LIN {X 0,Y 279.122,Z 639.162,A -85,B 0,C 180,E1 -18844.948,E2 -18844.948} C_VEL
LIN {X 0,Y 285.819,Z 626.252,A -85,B 0,C 180,E1 -18847.044,E2 -18847.044} C_VEL
LIN {X 0,Y 292.614,Z 612.071,A -85,B 0,C 180,E1 -18848.864,E2 -18848.864} C_VEL
LIN {X 0,Y 299.456,Z 596.451,A -85,B 0,C 180,E1 -18850.417,E2 -18850.417} C_VEL
LIN {X 0,Y 305.025,Z 582.195,A -85,B 0,C 180,E1 -18851.485,E2 -18851.485} C_VEL
LIN {X 0,Y 310.133,Z 566.91,A -85,B 0,C 180,E1 -18852.39,E2 -18852.39} C_VEL
LIN {X 0,Y 315.424,Z 547.486,A -85,B 0,C 180,E1 -18853.247,E2 -18853.247} C_VEL
LIN {X 0,Y 330.429,Z 486.43,A -85,B 0,C 180,E1 -18855.632,E2 -18855.632} C_VEL
LIN {X 0,Y 330.312,Z 486.665,A -85,B 0,C 180,E1 -18857.244,E2 -18857.244} C_VEL
LIN {X 0,Y 313.368,Z 553.571,A -85,B 0,C 180,E1 -18860.061,E2 -18860.061} C_VEL
LIN {X 0,Y 309.554,Z 566.236,A -85,B 0,C 180,E1 -18860.738,E2 -18860.738} C_VEL
LIN {X 0,Y 304.046,Z 581.734,A -85,B 0,C 180,E1 -18861.849,E2 -18861.849} C_VEL
LIN {X 0,Y 298.06,Z 596.489,A -85,B 0,C 180,E1 -18863.25,E2 -18863.25} C_VEL
LIN {X 0,Y 292.263,Z 609.131,A -85,B 0,C 180,E1 -18864.752,E2 -18864.752} C_VEL
LIN {X 0,Y 286.298,Z 620.873,A -85,B 0,C 180,E1 -18866.473,E2 -18866.473} C_VEL
LIN {X 0,Y 279.847,Z 632.628,A -85,B 0,C 180,E1 -18868.635,E2 -18868.635} C_VEL
LIN {X 0,Y 273.436,Z 643.529,A -85,B 0,C 180,E1 -18871.189,E2 -18871.189} C_VEL
LIN {X 0,Y 267.673,Z 652.584,A -85,B 0,C 180,E1 -18873.91,E2 -18873.91} C_VEL
LIN {X 0,Y 263.097,Z 659.179,A -85,B 0,C 180,E1 -18876.379,E2 -18876.379} C_VEL
LIN {X 0,Y 258.649,Z 665.21,A -85,B 0,C 180,E1 -18879.315,E2 -18879.315} C_VEL
LIN {X 0,Y 255.015,Z 669.8,A -85,B 0,C 180,E1 -18882.353,E2 -18882.353} C_VEL
LIN {X 0,Y 252.199,Z 673.017,A -85,B 0,C 180,E1 -18885.475,E2 -18885.475} C_VEL
LIN {X 0,Y 250.06,Z 674.932,A -85,B 0,C 180,E1 -18888.654,E2 -18888.654} C_VEL
LIN {X 0,Y 248.52,Z 675.55,A -85,B 0,C 180,E1 -18891.871,E2 -18891.871} C_VEL
LIN {X 0,Y 247.631,Z 674.837,A -85,B 0,C 180,E1 -18895.116,E2 -18895.116} C_VEL
LIN {X 0,Y 247.2,Z 672.768,A -85,B 0,C 180,E1 -18898.371,E2 -18898.371} C_VEL
LIN {X 0,Y 247.103,Z 669.276,A -85,B 0,C 180,E1 -18901.63,E2 -18901.63} C_VEL
LIN {X 0,Y 247.107,Z 665.658,A -85,B 0,C 180,E1 -18904.078,E2 -18904.078} C_VEL
LIN {X 0,Y 247.454,Z 659.333,A -85,B 0,C 180,E1 -18907.343,E2 -18907.343} C_VEL
LIN {X 0,Y 247.942,Z 652.241,A -85,B 0,C 180,E1 -18910.204,E2 -18910.204} C_VEL
LIN {X 0,Y 248.776,Z 643.485,A -85,B 0,C 180,E1 -18913.062,E2 -18913.062} C_VEL
LIN {X 0,Y 249.849,Z 634.415,A -85,B 0,C 180,E1 -18915.499,E2 -18915.499} C_VEL
LIN {X 0,Y 251.203,Z 623.335,A -85,B 0,C 180,E1 -18917.966,E2 -18917.966} C_VEL
LIN {X 0,Y 252.63,Z 611.516,A -85,B 0,C 180,E1 -18920.137,E2 -18920.137} C_VEL
LIN {X 0,Y 254.248,Z 598.401,A -85,B 0,C 180,E1 -18922.125,E2 -18922.125} C_VEL
LIN {X 0,Y 255.806,Z 585.81,A -85,B 0,C 180,E1 -18923.691,E2 -18923.691} C_VEL
LIN {X 0,Y 257.309,Z 571.28,A -85,B 0,C 180,E1 -18925.155,E2 -18925.155} C_VEL
LIN {X 0,Y 258.67,Z 555.661,A -85,B 0,C 180,E1 -18926.361,E2 -18926.361} C_VEL
LIN {X 0,Y 259.846,Z 539.566,A -85,B 0,C 180,E1 -18927.263,E2 -18927.263} C_VEL
LIN {X 0,Y 265.823,Z 443.881,A -85,B 0,C 180,E1 -18931.363,E2 -18931.363} C_VEL
LIN {X 0,Y 262.638,Z 420.691,A -85,B 0,C 180,E1 -18932.7,E2 -18932.7} C_VEL
LIN {X 0,Y 254.847,Z 398.323,A -85,B 0,C 180,E1 -18934.485,E2 -18934.485} C_VEL
LIN {X 0,Y 252.265,Z 387.318,A -85,B 0,C 180,E1 -18937.963,E2 -18937.963} C_VEL
LIN {X 0,Y 252.455,Z 387.301,A -85,B 0,C 180,E1 -18938.387,E2 -18938.387} C_VEL
LIN {X 0,Y 254.663,Z 388.809,A -85,B 0,C 180,E1 -18939.401,E2 -18939.401} C_VEL
LIN {X 0,Y 256.067,Z 390.357,A -85,B 0,C 180,E1 -18940.164,E2 -18940.164} C_VEL
LIN {X 0,Y 258.345,Z 395.76,A -85,B 0,C 180,E1 -18941.984,E2 -18941.984} C_VEL
LIN {X 0,Y 265.426,Z 407.166,A -85,B 0,C 180,E1 -18944.104,E2 -18944.104} C_VEL
LIN {X 0,Y 272.266,Z 419.25,A -85,B 0,C 180,E1 -18946.001,E2 -18946.001} C_VEL
LIN {X 0,Y 278.453,Z 431.445,A -85,B 0,C 180,E1 -18947.632,E2 -18947.632} C_VEL
LIN {X 0,Y 284.463,Z 445.002,A -85,B 0,C 180,E1 -18949.167,E2 -18949.167} C_VEL
LIN {X 0,Y 285.13,Z 447.431,A -85,B 0,C 180,E1 -18949.361,E2 -18949.361} C_VEL
LIN {X 0,Y 285.914,Z 453.843,A -85,B 0,C 180,E1 -18949.703,E2 -18949.703} C_VEL
LIN {X 0,Y 280.683,Z 561.87,A -85,B 0,C 180,E1 -18952.33,E2 -18952.33} C_VEL
LIN {X 0,Y 279.274,Z 577.479,A -85,B 0,C 180,E1 -18952.902,E2 -18952.902} C_VEL
LIN {X 0,Y 277.366,Z 591.845,A -85,B 0,C 180,E1 -18953.68,E2 -18953.68} C_VEL
LIN {X 0,Y 275.035,Z 605.926,A -85,B 0,C 180,E1 -18954.724,E2 -18954.724} C_VEL
LIN {X 0,Y 272.571,Z 618.27,A -85,B 0,C 180,E1 -18955.888,E2 -18955.888} C_VEL
LIN {X 0,Y 269.432,Z 631.557,A -85,B 0,C 180,E1 -18957.453,E2 -18957.453} C_VEL
LIN {X 0,Y 265.837,Z 644.861,A -85,B 0,C 180,E1 -18959.408,E2 -18959.408} C_VEL
LIN {X 0,Y 262.248,Z 656.841,A -85,B 0,C 180,E1 -18961.596,E2 -18961.596} C_VEL
LIN {X 0,Y 259.213,Z 666.822,A -85,B 0,C 180,E1 -18963.836,E2 -18963.836} C_VEL
LIN {X 0,Y 255.926,Z 676.732,A -85,B 0,C 180,E1 -18966.535,E2 -18966.535} C_VEL
LIN {X 0,Y 253.233,Z 684.89,A -85,B 0,C 180,E1 -18969.277,E2 -18969.277} C_VEL
LIN {X 0,Y 250.896,Z 692.062,A -85,B 0,C 180,E1 -18972.25,E2 -18972.25} C_VEL
LIN {X 0,Y 249.241,Z 697.898,A -85,B 0,C 180,E1 -18975.299,E2 -18975.299} C_VEL
LIN {X 0,Y 247.924,Z 702.738,A -85,B 0,C 180,E1 -18978.554,E2 -18978.554} C_VEL
LIN {X 0,Y 247.181,Z 706.288,A -85,B 0,C 180,E1 -18981.827,E2 -18981.827} C_VEL
LIN {X 0,Y 246.84,Z 708.688,A -85,B 0,C 180,E1 -18985.219,E2 -18985.219} C_VEL
LIN {X 0,Y 246.853,Z 709.819,A -85,B 0,C 180,E1 -18988.368,E2 -18988.368} C_VEL
LIN {X 0,Y 246.854,Z 709.83,A -85,B 0,C 180,E1 -18991.631,E2 -18991.631} C_VEL
LIN {X 0,Y 246.846,Z 708.687,A -85,B 0,C 180,E1 -18994.9,E2 -18994.9} C_VEL
LIN {X 0,Y 247.18,Z 706.393,A -85,B 0,C 180,E1 -18998.173,E2 -18998.173} C_VEL
LIN {X 0,Y 247.908,Z 702.898,A -85,B 0,C 180,E1 -19001.446,E2 -19001.446} C_VEL
LIN {X 0,Y 249.211,Z 698.113,A -85,B 0,C 180,E1 -19004.703,E2 -19004.703} C_VEL
LIN {X 0,Y 250.995,Z 691.907,A -85,B 0,C 180,E1 -19007.939,E2 -19007.939} C_VEL
LIN {X 0,Y 253.499,Z 684.109,A -85,B 0,C 180,E1 -19011.125,E2 -19011.125} C_VEL
LIN {X 0,Y 256.281,Z 675.796,A -85,B 0,C 180,E1 -19013.859,E2 -19013.859} C_VEL
LIN {X 0,Y 259.055,Z 667.491,A -85,B 0,C 180,E1 -19016.118,E2 -19016.118} C_VEL
LIN {X 0,Y 262.148,Z 657.361,A -85,B 0,C 180,E1 -19018.415,E2 -19018.415} C_VEL
LIN {X 0,Y 265.744,Z 645.49,A -85,B 0,C 180,E1 -19020.603,E2 -19020.603} C_VEL
LIN {X 0,Y 268.954,Z 633.613,A -85,B 0,C 180,E1 -19022.39,E2 -19022.39} C_VEL
LIN {X 0,Y 272.096,Z 620.752,A -85,B 0,C 180,E1 -19023.956,E2 -19023.956} C_VEL
LIN {X 0,Y 274.884,Z 607.255,A -85,B 0,C 180,E1 -19025.275,E2 -19025.275} C_VEL
LIN {X 0,Y 277.193,Z 593.324,A -85,B 0,C 180,E1 -19026.345,E2 -19026.345} C_VEL
LIN {X 0,Y 279.272,Z 578.654,A -85,B 0,C 180,E1 -19027.155,E2 -19027.155} C_VEL
LIN {X 0,Y 280.657,Z 563.713,A -85,B 0,C 180,E1 -19027.73,E2 -19027.73} C_VEL
LIN {X 0,Y 284.824,Z 478.026,A -85,B 0,C 180,E1 -19029.833,E2 -19029.833} C_VEL
LIN {X 0,Y 285.995,Z 452.937,A -85,B 0,C 180,E1 -19030.445,E2 -19030.445} C_VEL
LIN {X 0,Y 284.792,Z 445.554,A -85,B 0,C 180,E1 -19030.892,E2 -19030.892} C_VEL
LIN {X 0,Y 277.817,Z 429.915,A -85,B 0,C 180,E1 -19032.679,E2 -19032.679} C_VEL
LIN {X 0,Y 271.176,Z 417.234,A -85,B 0,C 180,E1 -19034.438,E2 -19034.438} C_VEL
LIN {X 0,Y 266.905,Z 409.496,A -85,B 0,C 180,E1 -19035.63,E2 -19035.63} C_VEL
LIN {X 0,Y 262.844,Z 404.965,A -85,B 0,C 180,E1 -19036.739,E2 -19036.739} C_VEL
LIN {X 0,Y 251.385,Z 395.568,A -85,B 0,C 180,E1 -19040.001,E2 -19040.001} C_VEL
LIN {X 0,Y 250.424,Z 394.069,A -85,B 0,C 180,E1 -19040.529,E2 -19040.529} C_VEL
LIN {X 0,Y 246.627,Z 385.224,A -85,B 0,C 180,E1 -19044.026,E2 -19044.026} C_VEL
LIN {X 0,Y 243.811,Z 378.951,A -85,B 0,C 180,E1 -19046.791,E2 -19046.791} C_VEL
LIN {X 0,Y 242.118,Z 375.757,A -85,B 0,C 180,E1 -19048.382,E2 -19048.382} C_VEL
LIN {X 0,Y 241.964,Z 374.965,A -85,B 0,C 180,E1 -19048.965,E2 -19048.965} C_VEL
LIN {X 0,Y 241.968,Z 374.95,A -85,B 0,C 180,E1 -19052.307,E2 -19052.307} C_VEL
LIN {X 0,Y 242.024,Z 374.953,A -85,B 0,C 180,E1 -19056.012,E2 -19056.012} C_VEL
LIN {X 0,Y 242.023,Z 374.952,A -85,B 0,C 180,E1 -19059.606,E2 -19059.606} C_VEL
LIN {X 0,Y 242.116,Z 374.923,A -85,B 0,C 180,E1 -19063.316,E2 -19063.316} C_VEL
LIN {X 0,Y 242.14,Z 374.946,A -85,B 0,C 180,E1 -19066.573,E2 -19066.573} C_VEL
LIN {X 0,Y 242.394,Z 374.914,A -85,B 0,C 180,E1 -19071.664,E2 -19071.664} C_VEL
LIN {X 0,Y 242.416,Z 374.898,A -85,B 0,C 180,E1 -19073.34,E2 -19073.34} C_VEL
LIN {X 0,Y 242.632,Z 374.888,A -85,B 0,C 180,E1 -19078.34,E2 -19078.34} C_VEL
LIN {X 0,Y 242.634,Z 374.854,A -85,B 0,C 180,E1 -19081.66,E2 -19081.66} C_VEL
LIN {X 0,Y 242.402,Z 374.888,A -85,B 0,C 180,E1 -19086.66,E2 -19086.66} C_VEL
LIN {X 0,Y 242.266,Z 374.922,A -85,B 0,C 180,E1 -19090.024,E2 -19090.024} C_VEL
LIN {X 0,Y 242.136,Z 374.925,A -85,B 0,C 180,E1 -19095.143,E2 -19095.143} C_VEL
LIN {X 0,Y 242.055,Z 374.935,A -85,B 0,C 180,E1 -19098.625,E2 -19098.625} C_VEL
LIN {X 0,Y 242.041,Z 374.961,A -85,B 0,C 180,E1 -19102.177,E2 -19102.177} C_VEL
LIN {X 0,Y 242.067,Z 374.937,A -85,B 0,C 180,E1 -19105.838,E2 -19105.838} C_VEL
LIN {X 0,Y 242.007,Z 374.945,A -85,B 0,C 180,E1 -19109.583,E2 -19109.583} C_VEL
LIN {X 0,Y 242.024,Z 375.2,A -85,B 0,C 180,E1 -19113.86,E2 -19113.86} C_VEL
LIN {X 0,Y 242.366,Z 376.481,A -85,B 0,C 180,E1 -19114.433,E2 -19114.433} C_VEL
LIN {X 0,Y 243.521,Z 378.521,A -85,B 0,C 180,E1 -19115.254,E2 -19115.254} C_VEL
LIN {X 0,Y 244.558,Z 379.622,A -85,B 0,C 180,E1 -19115.819,E2 -19115.819} C_VEL
LIN {X 0,Y 246.086,Z 382.714,A -85,B 0,C 180,E1 -19116.903,E2 -19116.903} C_VEL
LIN {X 0,Y 247.924,Z 385.881,A -85,B 0,C 180,E1 -19118.064,E2 -19118.064} C_VEL
LIN {X 0,Y 252.022,Z 392.901,A -85,B 0,C 180,E1 -19120.418,E2 -19120.418} C_VEL
LIN {X 0,Y 262.696,Z 408.315,A -85,B 0,C 180,E1 -19123.697,E2 -19123.697} C_VEL
LIN {X 0,Y 266.239,Z 414.331,A -85,B 0,C 180,E1 -19124.72,E2 -19124.72} C_VEL
LIN {X 0,Y 274.832,Z 434.1,A -85,B 0,C 180,E1 -19127.205,E2 -19127.205} C_VEL
LIN {X 0,Y 279.759,Z 446.521,A -85,B 0,C 180,E1 -19128.555,E2 -19128.555} C_VEL
LIN {X 0,Y 280.201,Z 450.816,A -85,B 0,C 180,E1 -19128.778,E2 -19128.778} C_VEL
LIN {X 0,Y 274.442,Z 565.143,A -85,B 0,C 180,E1 -19131.611,E2 -19131.611} C_VEL
LIN {X 0,Y 272.785,Z 581.258,A -85,B 0,C 180,E1 -19132.274,E2 -19132.274} C_VEL
LIN {X 0,Y 270.55,Z 596.378,A -85,B 0,C 180,E1 -19133.196,E2 -19133.196} C_VEL
LIN {X 0,Y 267.876,Z 610.662,A -85,B 0,C 180,E1 -19134.373,E2 -19134.373} C_VEL
LIN {X 0,Y 264.707,Z 624.939,A -85,B 0,C 180,E1 -19135.907,E2 -19135.907} C_VEL
LIN {X 0,Y 261.184,Z 638.082,A -85,B 0,C 180,E1 -19137.67,E2 -19137.67} C_VEL
LIN {X 0,Y 257.692,Z 650.157,A -85,B 0,C 180,E1 -19139.699,E2 -19139.699} C_VEL
LIN {X 0,Y 254.17,Z 661.17,A -85,B 0,C 180,E1 -19141.962,E2 -19141.962} C_VEL
LIN {X 0,Y 251.192,Z 670.446,A -85,B 0,C 180,E1 -19144.3,E2 -19144.3} C_VEL
LIN {X 0,Y 247.996,Z 679.538,A -85,B 0,C 180,E1 -19147.067,E2 -19147.067} C_VEL
LIN {X 0,Y 245.393,Z 687.077,A -85,B 0,C 180,E1 -19149.899,E2 -19149.899} C_VEL
LIN {X 0,Y 243.117,Z 694.112,A -85,B 0,C 180,E1 -19153.197,E2 -19153.197} C_VEL
LIN {X 0,Y 241.463,Z 699.634,A -85,B 0,C 180,E1 -19156.535,E2 -19156.535} C_VEL
LIN {X 0,Y 240.464,Z 703.796,A -85,B 0,C 180,E1 -19159.901,E2 -19159.901} C_VEL
LIN {X 0,Y 239.896,Z 706.71,A -85,B 0,C 180,E1 -19163.271,E2 -19163.271} C_VEL
LIN {X 0,Y 239.747,Z 708.446,A -85,B 0,C 180,E1 -19166.639,E2 -19166.639} C_VEL
LIN {X 0,Y 239.771,Z 709.037,A -85,B 0,C 180,E1 -19170,E2 -19170} C_VEL
LIN {X 0,Y 239.747,Z 708.439,A -85,B 0,C 180,E1 -19173.361,E2 -19173.361} C_VEL
LIN {X 0,Y 239.896,Z 706.691,A -85,B 0,C 180,E1 -19176.73,E2 -19176.73} C_VEL
LIN {X 0,Y 240.465,Z 703.759,A -85,B 0,C 180,E1 -19180.1,E2 -19180.1} C_VEL
LIN {X 0,Y 241.468,Z 699.576,A -85,B 0,C 180,E1 -19183.465,E2 -19183.465} C_VEL
LIN {X 0,Y 243.116,Z 694.041,A -85,B 0,C 180,E1 -19186.803,E2 -19186.803} C_VEL
LIN {X 0,Y 245.406,Z 687.021,A -85,B 0,C 180,E1 -19190.1,E2 -19190.1} C_VEL
LIN {X 0,Y 246.126,Z 685.348,A -85,B 0,C 180,E1 -19190.912,E2 -19190.912} C_VEL
LIN {X 0,Y 249.722,Z 679.837,A -85,B 0,C 180,E1 -19194.084,E2 -19194.084} C_VEL
LIN {X 0,Y 254.219,Z 673.05,A -85,B 0,C 180,E1 -19197.139,E2 -19197.139} C_VEL
LIN {X 0,Y 259.484,Z 664.907,A -85,B 0,C 180,E1 -19200.07,E2 -19200.07} C_VEL
LIN {X 0,Y 265.729,Z 655.198,A -85,B 0,C 180,E1 -19202.833,E2 -19202.833} C_VEL
LIN {X 0,Y 271.826,Z 645.226,A -85,B 0,C 180,E1 -19205.119,E2 -19205.119} C_VEL
LIN {X 0,Y 278.575,Z 633.661,A -85,B 0,C 180,E1 -19207.264,E2 -19207.264} C_VEL
LIN {X 0,Y 285.415,Z 621.131,A -85,B 0,C 180,E1 -19209.123,E2 -19209.123} C_VEL
LIN {X 0,Y 291.668,Z 608.732,A -85,B 0,C 180,E1 -19210.586,E2 -19210.586} C_VEL
LIN {X 0,Y 297.682,Z 595.659,A -85,B 0,C 180,E1 -19211.833,E2 -19211.833} C_VEL
LIN {X 0,Y 304.159,Z 579.833,A -85,B 0,C 180,E1 -19212.972,E2 -19212.972} C_VEL
LIN {X 0,Y 308.884,Z 566.463,A -85,B 0,C 180,E1 -19213.719,E2 -19213.719} C_VEL
LIN {X 0,Y 314.376,Z 547.514,A -85,B 0,C 180,E1 -19214.54,E2 -19214.54} C_VEL
LIN {X 0,Y 326.733,Z 499.697,A -85,B 0,C 180,E1 -19216.397,E2 -19216.397} C_VEL
LIN {X 0,Y 326.697,Z 499.799,A -85,B 0,C 180,E1 -19216.497,E2 -19216.497} C_VEL
LIN {X 0,Y 312.396,Z 553.674,A -85,B 0,C 180,E1 -19218.743,E2 -19218.743} C_VEL
LIN {X 0,Y 308.018,Z 567.356,A -85,B 0,C 180,E1 -19219.464,E2 -19219.464} C_VEL
LIN {X 0,Y 301.857,Z 583.519,A -85,B 0,C 180,E1 -19220.621,E2 -19220.621} C_VEL
LIN {X 0,Y 295.443,Z 598.066,A -85,B 0,C 180,E1 -19222.011,E2 -19222.011} C_VEL
LIN {X 0,Y 289.322,Z 610.357,A -85,B 0,C 180,E1 -19223.478,E2 -19223.478} C_VEL
LIN {X 0,Y 283.018,Z 621.864,A -85,B 0,C 180,E1 -19225.17,E2 -19225.17} C_VEL
LIN {X 0,Y 276.256,Z 633.219,A -85,B 0,C 180,E1 -19227.275,E2 -19227.275} C_VEL
LIN {X 0,Y 269.745,Z 643.456,A -85,B 0,C 180,E1 -19229.682,E2 -19229.682} C_VEL
LIN {X 0,Y 263.842,Z 652.028,A -85,B 0,C 180,E1 -19232.216,E2 -19232.216} C_VEL
LIN {X 0,Y 258.191,Z 659.57,A -85,B 0,C 180,E1 -19235.045,E2 -19235.045} C_VEL
LIN {X 0,Y 254.404,Z 664.223,A -85,B 0,C 180,E1 -19237.247,E2 -19237.247} C_VEL
LIN {X 0,Y 250.232,Z 669.141,A -85,B 0,C 180,E1 -19240.304,E2 -19240.304} C_VEL
LIN {X 0,Y 246.773,Z 672.719,A -85,B 0,C 180,E1 -19243.454,E2 -19243.454} C_VEL
LIN {X 0,Y 244.222,Z 674.978,A -85,B 0,C 180,E1 -19246.69,E2 -19246.69} C_VEL
LIN {X 0,Y 242.226,Z 675.982,A -85,B 0,C 180,E1 -19249.975,E2 -19249.975} C_VEL
LIN {X 0,Y 240.932,Z 675.682,A -85,B 0,C 180,E1 -19253.3,E2 -19253.3} C_VEL
LIN {X 0,Y 240.321,Z 674.056,A -85,B 0,C 180,E1 -19256.647,E2 -19256.647} C_VEL
LIN {X 0,Y 240.024,Z 671.057,A -85,B 0,C 180,E1 -19260,E2 -19260} C_VEL
LIN {X 0,Y 240.004,Z 667.817,A -85,B 0,C 180,E1 -19262.518,E2 -19262.518} C_VEL
LIN {X 0,Y 240.136,Z 662.471,A -85,B 0,C 180,E1 -19265.689,E2 -19265.689} C_VEL
LIN {X 0,Y 240.503,Z 656.646,A -85,B 0,C 180,E1 -19268.402,E2 -19268.402} C_VEL
LIN {X 0,Y 241.167,Z 648.83,A -85,B 0,C 180,E1 -19271.345,E2 -19271.345} C_VEL
LIN {X 0,Y 242.188,Z 639.234,A -85,B 0,C 180,E1 -19274.28,E2 -19274.28} C_VEL
LIN {X 0,Y 243.385,Z 629.266,A -85,B 0,C 180,E1 -19276.784,E2 -19276.784} C_VEL
LIN {X 0,Y 244.885,Z 617.238,A -85,B 0,C 180,E1 -19279.271,E2 -19279.271} C_VEL
LIN {X 0,Y 246.533,Z 603.914,A -85,B 0,C 180,E1 -19281.533,E2 -19281.533} C_VEL
LIN {X 0,Y 248.23,Z 590.761,A -85,B 0,C 180,E1 -19283.352,E2 -19283.352} C_VEL
LIN {X 0,Y 249.862,Z 576.362,A -85,B 0,C 180,E1 -19284.956,E2 -19284.956} C_VEL
LIN {X 0,Y 251.312,Z 560.95,A -85,B 0,C 180,E1 -19286.3,E2 -19286.3} C_VEL
LIN {X 0,Y 252.568,Z 545.22,A -85,B 0,C 180,E1 -19287.33,E2 -19287.33} C_VEL
LIN {X 0,Y 259.073,Z 444.798,A -85,B 0,C 180,E1 -19291.821,E2 -19291.821} C_VEL
LIN {X 0,Y 256.233,Z 423.114,A -85,B 0,C 180,E1 -19293.104,E2 -19293.104} C_VEL
LIN {X 0,Y 247.62,Z 398.369,A -85,B 0,C 180,E1 -19295.139,E2 -19295.139} C_VEL
LIN {X 0,Y 246.029,Z 391.561,A -85,B 0,C 180,E1 -19297.369,E2 -19297.369} C_VEL
LIN {X 0,Y 246.194,Z 391.53,A -85,B 0,C 180,E1 -19297.718,E2 -19297.718} C_VEL
LIN {X 0,Y 250.812,Z 395.097,A -85,B 0,C 180,E1 -19299.969,E2 -19299.969} C_VEL
LIN {X 0,Y 256.069,Z 403.369,A -85,B 0,C 180,E1 -19301.753,E2 -19301.753} C_VEL
LIN {X 0,Y 262.245,Z 413.431,A -85,B 0,C 180,E1 -19303.63,E2 -19303.63} C_VEL
LIN {X 0,Y 269.596,Z 426.891,A -85,B 0,C 180,E1 -19305.731,E2 -19305.731} C_VEL
LIN {X 0,Y 275.983,Z 440.167,A -85,B 0,C 180,E1 -19307.466,E2 -19307.466} C_VEL
LIN {X 0,Y 279.779,Z 449.148,A -85,B 0,C 180,E1 -19308.475,E2 -19308.475} C_VEL
LIN {X 0,Y 280.459,Z 455.36,A -85,B 0,C 180,E1 -19308.805,E2 -19308.805} C_VEL
LIN {X 0,Y 274.99,Z 563.173,A -85,B 0,C 180,E1 -19311.467,E2 -19311.467} C_VEL
LIN {X 0,Y 273.446,Z 579.168,A -85,B 0,C 180,E1 -19312.089,E2 -19312.089} C_VEL
LIN {X 0,Y 271.277,Z 594.318,A -85,B 0,C 180,E1 -19312.962,E2 -19312.962} C_VEL
LIN {X 0,Y 268.722,Z 608.521,A -85,B 0,C 180,E1 -19314.081,E2 -19314.081} C_VEL
LIN {X 0,Y 265.988,Z 621.373,A -85,B 0,C 180,E1 -19315.383,E2 -19315.383} C_VEL
LIN {X 0,Y 262.741,Z 634.108,A -85,B 0,C 180,E1 -19316.975,E2 -19316.975} C_VEL
LIN {X 0,Y 259.068,Z 646.947,A -85,B 0,C 180,E1 -19318.973,E2 -19318.973} C_VEL
LIN {X 0,Y 255.405,Z 658.581,A -85,B 0,C 180,E1 -19321.213,E2 -19321.213} C_VEL
LIN {X 0,Y 252.316,Z 668.371,A -85,B 0,C 180,E1 -19323.534,E2 -19323.534} C_VEL
LIN {X 0,Y 248.932,Z 677.945,A -85,B 0,C 180,E1 -19326.277,E2 -19326.277} C_VEL
LIN {X 0,Y 246.193,Z 685.921,A -85,B 0,C 180,E1 -19329.094,E2 -19329.094} C_VEL
LIN {X 0,Y 243.742,Z 693.185,A -85,B 0,C 180,E1 -19332.288,E2 -19332.288} C_VEL
LIN {X 0,Y 241.929,Z 699.242,A -85,B 0,C 180,E1 -19335.704,E2 -19335.704} C_VEL
LIN {X 0,Y 240.928,Z 702.724,A -85,B 0,C 180,E1 -19338.217,E2 -19338.217} C_VEL
LIN {X 0,Y 240.138,Z 706.275,A -85,B 0,C 180,E1 -19341.585,E2 -19341.585} C_VEL
LIN {X 0,Y 239.768,Z 708.617,A -85,B 0,C 180,E1 -19344.955,E2 -19344.955} C_VEL
LIN {X 0,Y 239.748,Z 709.805,A -85,B 0,C 180,E1 -19348.32,E2 -19348.32} C_VEL
LIN {X 0,Y 239.748,Z 709.816,A -85,B 0,C 180,E1 -19351.68,E2 -19351.68} C_VEL
LIN {X 0,Y 239.767,Z 708.672,A -85,B 0,C 180,E1 -19355.045,E2 -19355.045} C_VEL
LIN {X 0,Y 240.138,Z 706.378,A -85,B 0,C 180,E1 -19358.414,E2 -19358.414} C_VEL
LIN {X 0,Y 240.912,Z 702.883,A -85,B 0,C 180,E1 -19361.783,E2 -19361.783} C_VEL
LIN {X 0,Y 242.305,Z 698.096,A -85,B 0,C 180,E1 -19365.132,E2 -19365.132} C_VEL
LIN {X 0,Y 244.21,Z 691.89,A -85,B 0,C 180,E1 -19368.455,E2 -19368.455} C_VEL
LIN {X 0,Y 246.849,Z 684.091,A -85,B 0,C 180,E1 -19371.723,E2 -19371.723} C_VEL
LIN {X 0,Y 249.778,Z 675.776,A -85,B 0,C 180,E1 -19374.52,E2 -19374.52} C_VEL
LIN {X 0,Y 252.893,Z 666.637,A -85,B 0,C 180,E1 -19377.047,E2 -19377.047} C_VEL
LIN {X 0,Y 256.467,Z 655.513,A -85,B 0,C 180,E1 -19379.555,E2 -19379.555} C_VEL
LIN {X 0,Y 260.25,Z 643.243,A -85,B 0,C 180,E1 -19381.775,E2 -19381.775} C_VEL
LIN {X 0,Y 263.688,Z 630.954,A -85,B 0,C 180,E1 -19383.576,E2 -19383.576} C_VEL
LIN {X 0,Y 266.941,Z 617.523,A -85,B 0,C 180,E1 -19385.163,E2 -19385.163} C_VEL
LIN {X 0,Y 269.72,Z 603.955,A -85,B 0,C 180,E1 -19386.436,E2 -19386.436} C_VEL
LIN {X 0,Y 271.95,Z 590.762,A -85,B 0,C 180,E1 -19387.395,E2 -19387.395} C_VEL
LIN {X 0,Y 274.054,Z 575.084,A -85,B 0,C 180,E1 -19388.219,E2 -19388.219} C_VEL
LIN {X 0,Y 275.362,Z 559.364,A -85,B 0,C 180,E1 -19388.763,E2 -19388.763} C_VEL
LIN {X 0,Y 280.571,Z 455.16,A -85,B 0,C 180,E1 -19391.317,E2 -19391.317} C_VEL
LIN {X 0,Y 279.667,Z 448.556,A -85,B 0,C 180,E1 -19391.701,E2 -19391.701} C_VEL
LIN {X 0,Y 272.904,Z 433.33,A -85,B 0,C 180,E1 -19393.51,E2 -19393.51} C_VEL
LIN {X 0,Y 265.595,Z 419.231,A -85,B 0,C 180,E1 -19395.548,E2 -19395.548} C_VEL
LIN {X 0,Y 259.552,Z 408.881,A -85,B 0,C 180,E1 -19397.329,E2 -19397.329} C_VEL
LIN {X 0,Y 252.405,Z 397.638,A -85,B 0,C 180,E1 -19399.59,E2 -19399.59} C_VEL
LIN {X 0,Y 250.759,Z 394.914,A -85,B 0,C 180,E1 -19400.225,E2 -19400.225} C_VEL
LIN {X 0,Y 250.424,Z 394.069,A -85,B 0,C 180,E1 -19400.529,E2 -19400.529} C_VEL
LIN {X 0,Y 249.361,Z 392.245,A -85,B 0,C 180,E1 -19401.291,E2 -19401.291} C_VEL
LIN {X 0,Y 247.125,Z 390.261,A -85,B 0,C 180,E1 -19402.475,E2 -19402.475} C_VEL
LIN {X 0,Y 241.118,Z 386.858,A -85,B 0,C 180,E1 -19405.334,E2 -19405.334} C_VEL
LIN {X 0,Y 239.216,Z 384.804,A -85,B 0,C 180,E1 -19406.59,E2 -19406.59} C_VEL
LIN {X 0,Y 238.802,Z 383.917,A -85,B 0,C 180,E1 -19407.005,E2 -19407.005} C_VEL
LIN {X 0,Y 234.955,Z 376.108,A -85,B 0,C 180,E1 -19411.141,E2 -19411.141} C_VEL
LIN {X 0,Y 234.945,Z 375.823,A -85,B 0,C 180,E1 -19413.339,E2 -19413.339} C_VEL
LIN {X 0,Y 234.986,Z 375.814,A -85,B 0,C 180,E1 -19417.995,E2 -19417.995} C_VEL
LIN {X 0,Y 235.056,Z 375.802,A -85,B 0,C 180,E1 -19423.092,E2 -19423.092} C_VEL
LIN {X 0,Y 235.1,Z 375.8,A -85,B 0,C 180,E1 -19427.921,E2 -19427.921} C_VEL
LIN {X 0,Y 235.327,Z 375.79,A -85,B 0,C 180,E1 -19431.412,E2 -19431.412} C_VEL
LIN {X 0,Y 235.367,Z 375.778,A -85,B 0,C 180,E1 -19433.14,E2 -19433.14} C_VEL
LIN {X 0,Y 235.591,Z 375.765,A -85,B 0,C 180,E1 -19438.29,E2 -19438.29} C_VEL
LIN {X 0,Y 235.594,Z 375.731,A -85,B 0,C 180,E1 -19441.709,E2 -19441.709} C_VEL
LIN {X 0,Y 235.352,Z 375.763,A -85,B 0,C 180,E1 -19446.86,E2 -19446.86} C_VEL
LIN {X 0,Y 235.212,Z 375.805,A -85,B 0,C 180,E1 -19450.327,E2 -19450.327} C_VEL
LIN {X 0,Y 235.08,Z 375.809,A -85,B 0,C 180,E1 -19455.608,E2 -19455.608} C_VEL
LIN {X 0,Y 234.995,Z 375.81,A -85,B 0,C 180,E1 -19459.206,E2 -19459.206} C_VEL
LIN {X 0,Y 234.975,Z 375.836,A -85,B 0,C 180,E1 -19462.881,E2 -19462.881} C_VEL
LIN {X 0,Y 234.969,Z 375.829,A -85,B 0,C 180,E1 -19466.657,E2 -19466.657} C_VEL
LIN {X 0,Y 234.937,Z 375.956,A -85,B 0,C 180,E1 -19471.191,E2 -19471.191} C_VEL
LIN {X 0,Y 235.171,Z 377.004,A -85,B 0,C 180,E1 -19471.784,E2 -19471.784} C_VEL
LIN {X 0,Y 235.882,Z 378.597,A -85,B 0,C 180,E1 -19472.432,E2 -19472.432} C_VEL
LIN {X 0,Y 237.289,Z 380.284,A -85,B 0,C 180,E1 -19473.353,E2 -19473.353} C_VEL
LIN {X 0,Y 243.023,Z 390.234,A -85,B 0,C 180,E1 -19477.394,E2 -19477.394} C_VEL
LIN {X 0,Y 245.004,Z 393.522,A -85,B 0,C 180,E1 -19478.47,E2 -19478.47} C_VEL
LIN {X 0,Y 251.835,Z 402.908,A -85,B 0,C 180,E1 -19480.8,E2 -19480.8} C_VEL
LIN {X 0,Y 260.971,Z 416.733,A -85,B 0,C 180,E1 -19483.627,E2 -19483.627} C_VEL
LIN {X 0,Y 266.121,Z 428.208,A -85,B 0,C 180,E1 -19485.214,E2 -19485.214} C_VEL
LIN {X 0,Y 273.318,Z 445.92,A -85,B 0,C 180,E1 -19487.324,E2 -19487.324} C_VEL
LIN {X 0,Y 274.677,Z 449.56,A -85,B 0,C 180,E1 -19487.712,E2 -19487.712} C_VEL
LIN {X 0,Y 274.8,Z 453.039,A -85,B 0,C 180,E1 -19487.856,E2 -19487.856} C_VEL
LIN {X 0,Y 268.916,Z 565.259,A -85,B 0,C 180,E1 -19490.672,E2 -19490.672} C_VEL
LIN {X 0,Y 267.215,Z 581.325,A -85,B 0,C 180,E1 -19491.344,E2 -19491.344} C_VEL
LIN {X 0,Y 264.886,Z 596.427,A -85,B 0,C 180,E1 -19492.273,E2 -19492.273} C_VEL
LIN {X 0,Y 262.185,Z 610.373,A -85,B 0,C 180,E1 -19493.434,E2 -19493.434} C_VEL
LIN {X 0,Y 258.834,Z 625.061,A -85,B 0,C 180,E1 -19495.038,E2 -19495.038} C_VEL
LIN {X 0,Y 255.204,Z 638.11,A -85,B 0,C 180,E1 -19496.816,E2 -19496.816} C_VEL
LIN {X 0,Y 251.565,Z 650.181,A -85,B 0,C 180,E1 -19498.88,E2 -19498.88} C_VEL
LIN {X 0,Y 247.88,Z 661.192,A -85,B 0,C 180,E1 -19501.185,E2 -19501.185} C_VEL
LIN {X 0,Y 244.777,Z 670.466,A -85,B 0,C 180,E1 -19503.575,E2 -19503.575} C_VEL
LIN {X 0,Y 241.418,Z 679.556,A -85,B 0,C 180,E1 -19506.404,E2 -19506.404} C_VEL
LIN {X 0,Y 238.669,Z 687.095,A -85,B 0,C 180,E1 -19509.307,E2 -19509.307} C_VEL
LIN {X 0,Y 236.279,Z 694.128,A -85,B 0,C 180,E1 -19512.696,E2 -19512.696} C_VEL
LIN {X 0,Y 234.533,Z 699.65,A -85,B 0,C 180,E1 -19516.13,E2 -19516.13} C_VEL
LIN {X 0,Y 233.44,Z 703.811,A -85,B 0,C 180,E1 -19519.593,E2 -19519.593} C_VEL
LIN {X 0,Y 232.816,Z 706.724,A -85,B 0,C 180,E1 -19523.065,E2 -19523.065} C_VEL
LIN {X 0,Y 232.658,Z 708.46,A -85,B 0,C 180,E1 -19526.537,E2 -19526.537} C_VEL
LIN {X 0,Y 232.687,Z 709.051,A -85,B 0,C 180,E1 -19530,E2 -19530} C_VEL
LIN {X 0,Y 232.659,Z 708.452,A -85,B 0,C 180,E1 -19533.464,E2 -19533.464} C_VEL
LIN {X 0,Y 232.816,Z 706.704,A -85,B 0,C 180,E1 -19536.935,E2 -19536.935} C_VEL
LIN {X 0,Y 233.441,Z 703.773,A -85,B 0,C 180,E1 -19540.407,E2 -19540.407} C_VEL
LIN {X 0,Y 234.538,Z 699.59,A -85,B 0,C 180,E1 -19543.87,E2 -19543.87} C_VEL
LIN {X 0,Y 236.273,Z 694.055,A -85,B 0,C 180,E1 -19547.305,E2 -19547.305} C_VEL
LIN {X 0,Y 238.896,Z 686.711,A -85,B 0,C 180,E1 -19550.898,E2 -19550.898} C_VEL
LIN {X 0,Y 242.242,Z 682.109,A -85,B 0,C 180,E1 -19553.965,E2 -19553.965} C_VEL
LIN {X 0,Y 246.71,Z 676.018,A -85,B 0,C 180,E1 -19557.116,E2 -19557.116} C_VEL
LIN {X 0,Y 252.068,Z 668.637,A -85,B 0,C 180,E1 -19560.124,E2 -19560.124} C_VEL
LIN {X 0,Y 258.328,Z 659.841,A -85,B 0,C 180,E1 -19562.964,E2 -19562.964} C_VEL
LIN {X 0,Y 265.427,Z 649.442,A -85,B 0,C 180,E1 -19565.628,E2 -19565.628} C_VEL
LIN {X 0,Y 272.327,Z 638.784,A -85,B 0,C 180,E1 -19567.801,E2 -19567.801} C_VEL
LIN {X 0,Y 279.85,Z 626.411,A -85,B 0,C 180,E1 -19569.821,E2 -19569.821} C_VEL
LIN {X 0,Y 286.793,Z 614.022,A -85,B 0,C 180,E1 -19571.426,E2 -19571.426} C_VEL
LIN {X 0,Y 294.248,Z 599.405,A -85,B 0,C 180,E1 -19572.9,E2 -19572.9} C_VEL
LIN {X 0,Y 300.942,Z 584.674,A -85,B 0,C 180,E1 -19574.008,E2 -19574.008} C_VEL
LIN {X 0,Y 306.465,Z 570.665,A -85,B 0,C 180,E1 -19574.844,E2 -19574.844} C_VEL
LIN {X 0,Y 312.077,Z 553.733,A -85,B 0,C 180,E1 -19575.598,E2 -19575.598} C_VEL
LIN {X 0,Y 317.925,Z 532.036,A -85,B 0,C 180,E1 -19576.461,E2 -19576.461} C_VEL
LIN {X 0,Y 316.31,Z 537.919,A -85,B 0,C 180,E1 -19576.74,E2 -19576.74} C_VEL
LIN {X 0,Y 310.012,Z 559.733,A -85,B 0,C 180,E1 -19577.7,E2 -19577.7} C_VEL
LIN {X 0,Y 304.959,Z 573.641,A -85,B 0,C 180,E1 -19578.504,E2 -19578.504} C_VEL
LIN {X 0,Y 299.267,Z 587.033,A -85,B 0,C 180,E1 -19579.509,E2 -19579.509} C_VEL
LIN {X 0,Y 293.031,Z 599.956,A -85,B 0,C 180,E1 -19580.76,E2 -19580.76} C_VEL
LIN {X 0,Y 286.595,Z 611.894,A -85,B 0,C 180,E1 -19582.189,E2 -19582.189} C_VEL
LIN {X 0,Y 278.923,Z 624.779,A -85,B 0,C 180,E1 -19584.139,E2 -19584.139} C_VEL
LIN {X 0,Y 271.855,Z 635.647,A -85,B 0,C 180,E1 -19586.233,E2 -19586.233} C_VEL
LIN {X 0,Y 264.549,Z 646.005,A -85,B 0,C 180,E1 -19588.8,E2 -19588.8} C_VEL
LIN {X 0,Y 257.942,Z 654.61,A -85,B 0,C 180,E1 -19591.523,E2 -19591.523} C_VEL
LIN {X 0,Y 252.044,Z 661.683,A -85,B 0,C 180,E1 -19594.393,E2 -19594.393} C_VEL
LIN {X 0,Y 246.922,Z 667.292,A -85,B 0,C 180,E1 -19597.403,E2 -19597.403} C_VEL
LIN {X 0,Y 243.703,Z 670.582,A -85,B 0,C 180,E1 -19599.754,E2 -19599.754} C_VEL
LIN {X 0,Y 240.065,Z 673.828,A -85,B 0,C 180,E1 -19602.977,E2 -19602.977} C_VEL
LIN {X 0,Y 237.362,Z 675.797,A -85,B 0,C 180,E1 -19606.298,E2 -19606.298} C_VEL
LIN {X 0,Y 235.275,Z 676.526,A -85,B 0,C 180,E1 -19609.675,E2 -19609.675} C_VEL
LIN {X 0,Y 233.889,Z 675.965,A -85,B 0,C 180,E1 -19613.097,E2 -19613.097} C_VEL
LIN {X 0,Y 233.24,Z 674.086,A -85,B 0,C 180,E1 -19616.545,E2 -19616.545} C_VEL
LIN {X 0,Y 232.953,Z 670.828,A -85,B 0,C 180,E1 -19620,E2 -19620} C_VEL
LIN {X 0,Y 232.953,Z 666.063,A -85,B 0,C 180,E1 -19623.459,E2 -19623.459} C_VEL
LIN {X 0,Y 233.103,Z 661.617,A -85,B 0,C 180,E1 -19625.971,E2 -19625.971} C_VEL
LIN {X 0,Y 233.541,Z 654.705,A -85,B 0,C 180,E1 -19629.09,E2 -19629.09} C_VEL
LIN {X 0,Y 234.291,Z 646.339,A -85,B 0,C 180,E1 -19632.121,E2 -19632.121} C_VEL
LIN {X 0,Y 235.479,Z 636.074,A -85,B 0,C 180,E1 -19635.138,E2 -19635.138} C_VEL
LIN {X 0,Y 236.829,Z 624.772,A -85,B 0,C 180,E1 -19637.863,E2 -19637.863} C_VEL
LIN {X 0,Y 238.395,Z 612.581,A -85,B 0,C 180,E1 -19640.267,E2 -19640.267} C_VEL
LIN {X 0,Y 240.012,Z 599.563,A -85,B 0,C 180,E1 -19642.375,E2 -19642.375} C_VEL
LIN {X 0,Y 241.848,Z 585.454,A -85,B 0,C 180,E1 -19644.234,E2 -19644.234} C_VEL
LIN {X 0,Y 243.393,Z 570.877,A -85,B 0,C 180,E1 -19645.774,E2 -19645.774} C_VEL
LIN {X 0,Y 244.816,Z 555.11,A -85,B 0,C 180,E1 -19647.053,E2 -19647.053} C_VEL
LIN {X 0,Y 246.059,Z 539.031,A -85,B 0,C 180,E1 -19648.002,E2 -19648.002} C_VEL
LIN {X 0,Y 252.263,Z 445.137,A -85,B 0,C 180,E1 -19652.33,E2 -19652.33} C_VEL
LIN {X 0,Y 249.63,Z 425.077,A -85,B 0,C 180,E1 -19653.553,E2 -19653.553} C_VEL
LIN {X 0,Y 240.442,Z 398.773,A -85,B 0,C 180,E1 -19655.774,E2 -19655.774} C_VEL
LIN {X 0,Y 239.987,Z 396.742,A -85,B 0,C 180,E1 -19656.396,E2 -19656.396} C_VEL
LIN {X 0,Y 240.063,Z 396.459,A -85,B 0,C 180,E1 -19656.807,E2 -19656.807} C_VEL
LIN {X 0,Y 241.643,Z 397.463,A -85,B 0,C 180,E1 -19657.497,E2 -19657.497} C_VEL
LIN {X 0,Y 244.257,Z 398.771,A -85,B 0,C 180,E1 -19658.347,E2 -19658.347} C_VEL
LIN {X 0,Y 247.79,Z 401.266,A -85,B 0,C 180,E1 -19659.476,E2 -19659.476} C_VEL
LIN {X 0,Y 254.491,Z 411.875,A -85,B 0,C 180,E1 -19661.709,E2 -19661.709} C_VEL
LIN {X 0,Y 260.078,Z 421.478,A -85,B 0,C 180,E1 -19663.446,E2 -19663.446} C_VEL
LIN {X 0,Y 267.447,Z 435.63,A -85,B 0,C 180,E1 -19665.605,E2 -19665.605} C_VEL
LIN {X 0,Y 273.443,Z 449.057,A -85,B 0,C 180,E1 -19667.29,E2 -19667.29} C_VEL
LIN {X 0,Y 274.769,Z 452.794,A -85,B 0,C 180,E1 -19667.674,E2 -19667.674} C_VEL
LIN {X 0,Y 275.091,Z 456.466,A -85,B 0,C 180,E1 -19667.861,E2 -19667.861} C_VEL
LIN {X 0,Y 269.485,Z 563.094,A -85,B 0,C 180,E1 -19670.529,E2 -19670.529} C_VEL
LIN {X 0,Y 267.891,Z 579.119,A -85,B 0,C 180,E1 -19671.158,E2 -19671.158} C_VEL
LIN {X 0,Y 265.635,Z 594.281,A -85,B 0,C 180,E1 -19672.038,E2 -19672.038} C_VEL
LIN {X 0,Y 262.943,Z 608.731,A -85,B 0,C 180,E1 -19673.193,E2 -19673.193} C_VEL
LIN {X 0,Y 260.128,Z 621.523,A -85,B 0,C 180,E1 -19674.514,E2 -19674.514} C_VEL
LIN {X 0,Y 256.428,Z 635.354,A -85,B 0,C 180,E1 -19676.289,E2 -19676.289} C_VEL
LIN {X 0,Y 252.638,Z 647.982,A -85,B 0,C 180,E1 -19678.327,E2 -19678.327} C_VEL
LIN {X 0,Y 249.181,Z 658.564,A -85,B 0,C 180,E1 -19680.424,E2 -19680.424} C_VEL
LIN {X 0,Y 245.918,Z 668.355,A -85,B 0,C 180,E1 -19682.789,E2 -19682.789} C_VEL
LIN {X 0,Y 242.877,Z 676.701,A -85,B 0,C 180,E1 -19685.192,E2 -19685.192} C_VEL
LIN {X 0,Y 239.905,Z 684.861,A -85,B 0,C 180,E1 -19688.067,E2 -19688.067} C_VEL
LIN {X 0,Y 237.051,Z 692.814,A -85,B 0,C 180,E1 -19691.573,E2 -19691.573} C_VEL
LIN {X 0,Y 235.009,Z 699.228,A -85,B 0,C 180,E1 -19695.274,E2 -19695.274} C_VEL
LIN {X 0,Y 233.919,Z 702.71,A -85,B 0,C 180,E1 -19697.859,E2 -19697.859} C_VEL
LIN {X 0,Y 233.084,Z 706.261,A -85,B 0,C 180,E1 -19701.329,E2 -19701.329} C_VEL
LIN {X 0,Y 232.688,Z 708.604,A -85,B 0,C 180,E1 -19704.801,E2 -19704.801} C_VEL
LIN {X 0,Y 232.645,Z 709.791,A -85,B 0,C 180,E1 -19708.269,E2 -19708.269} C_VEL
LIN {X 0,Y 232.687,Z 709.948,A -85,B 0,C 180,E1 -19710,E2 -19710} C_VEL
LIN {X 0,Y 232.628,Z 709.372,A -85,B 0,C 180,E1 -19713.464,E2 -19713.464} C_VEL
LIN {X 0,Y 232.818,Z 707.657,A -85,B 0,C 180,E1 -19716.935,E2 -19716.935} C_VEL
LIN {X 0,Y 233.444,Z 704.77,A -85,B 0,C 180,E1 -19720.406,E2 -19720.406} C_VEL
LIN {X 0,Y 234.554,Z 700.642,A -85,B 0,C 180,E1 -19723.869,E2 -19723.869} C_VEL
LIN {X 0,Y 236.326,Z 695.164,A -85,B 0,C 180,E1 -19727.3,E2 -19727.3} C_VEL
LIN {X 0,Y 238.697,Z 688.186,A -85,B 0,C 180,E1 -19730.69,E2 -19730.69} C_VEL
LIN {X 0,Y 241.415,Z 680.715,A -85,B 0,C 180,E1 -19733.596,E2 -19733.596} C_VEL
LIN {X 0,Y 244.809,Z 671.715,A -85,B 0,C 180,E1 -19736.422,E2 -19736.422} C_VEL
LIN {X 0,Y 247.89,Z 662.518,A -85,B 0,C 180,E1 -19738.814,E2 -19738.814} C_VEL
LIN {X 0,Y 251.931,Z 650.68,A -85,B 0,C 180,E1 -19741.303,E2 -19741.303} C_VEL
LIN {X 0,Y 255.591,Z 638.599,A -85,B 0,C 180,E1 -19743.363,E2 -19743.363} C_VEL
LIN {X 0,Y 259.206,Z 625.678,A -85,B 0,C 180,E1 -19745.121,E2 -19745.121} C_VEL
LIN {X 0,Y 262.438,Z 611.695,A -85,B 0,C 180,E1 -19746.656,E2 -19746.656} C_VEL
LIN {X 0,Y 265.279,Z 596.975,A -85,B 0,C 180,E1 -19747.901,E2 -19747.901} C_VEL
LIN {X 0,Y 267.649,Z 581.988,A -85,B 0,C 180,E1 -19748.823,E2 -19748.823} C_VEL
LIN {X 0,Y 269.371,Z 566.246,A -85,B 0,C 180,E1 -19749.491,E2 -19749.491} C_VEL
LIN {X 0,Y 271.96,Z 520.071,A -85,B 0,C 180,E1 -19750.67,E2 -19750.67} C_VEL
LIN {X 0,Y 275.223,Z 455.3,A -85,B 0,C 180,E1 -19752.293,E2 -19752.293} C_VEL
LIN {X 0,Y 274.539,Z 451.466,A -85,B 0,C 180,E1 -19752.555,E2 -19752.555} C_VEL
LIN {X 0,Y 267.662,Z 435.923,A -85,B 0,C 180,E1 -19754.484,E2 -19754.484} C_VEL
LIN {X 0,Y 260.466,Z 422.125,A -85,B 0,C 180,E1 -19756.59,E2 -19756.59} C_VEL
LIN {X 0,Y 254.796,Z 412.373,A -85,B 0,C 180,E1 -19758.351,E2 -19758.351} C_VEL
LIN {X 0,Y 247.698,Z 401.046,A -85,B 0,C 180,E1 -19760.726,E2 -19760.726} C_VEL
LIN {X 0,Y 243.554,Z 394.778,A -85,B 0,C 180,E1 -19762.309,E2 -19762.309} C_VEL
LIN {X 0,Y 240.507,Z 387.76,A -85,B 0,C 180,E1 -19765.261,E2 -19765.261} C_VEL
LIN {X 0,Y 238.802,Z 383.917,A -85,B 0,C 180,E1 -19767.005,E2 -19767.005} C_VEL
LIN {X 0,Y 237.433,Z 381.561,A -85,B 0,C 180,E1 -19768.275,E2 -19768.275} C_VEL
LIN {X 0,Y 234.664,Z 379.587,A -85,B 0,C 180,E1 -19770.018,E2 -19770.018} C_VEL
LIN {X 0,Y 228.021,Z 377.022,A -85,B 0,C 180,E1 -19773.912,E2 -19773.912} C_VEL
LIN {X 0,Y 227.94,Z 376.875,A -85,B 0,C 180,E1 -19774.092,E2 -19774.092} C_VEL
LIN {X 0,Y 227.952,Z 376.69,A -85,B 0,C 180,E1 -19778.286,E2 -19778.286} C_VEL
LIN {X 0,Y 228.025,Z 376.679,A -85,B 0,C 180,E1 -19783.895,E2 -19783.895} C_VEL
LIN {X 0,Y 228.058,Z 376.681,A -85,B 0,C 180,E1 -19787.542,E2 -19787.542} C_VEL
LIN {X 0,Y 228.264,Z 376.664,A -85,B 0,C 180,E1 -19791.144,E2 -19791.144} C_VEL
LIN {X 0,Y 228.318,Z 376.659,A -85,B 0,C 180,E1 -19792.927,E2 -19792.927} C_VEL
LIN {X 0,Y 228.549,Z 376.642,A -85,B 0,C 180,E1 -19798.238,E2 -19798.238} C_VEL
LIN {X 0,Y 228.552,Z 376.607,A -85,B 0,C 180,E1 -19801.762,E2 -19801.762} C_VEL
LIN {X 0,Y 228.304,Z 376.639,A -85,B 0,C 180,E1 -19807.073,E2 -19807.073} C_VEL
LIN {X 0,Y 228.142,Z 376.689,A -85,B 0,C 180,E1 -19810.651,E2 -19810.651} C_VEL
LIN {X 0,Y 228.038,Z 376.672,A -85,B 0,C 180,E1 -19814.274,E2 -19814.274} C_VEL
LIN {X 0,Y 227.969,Z 376.696,A -85,B 0,C 180,E1 -19817.956,E2 -19817.956} C_VEL
LIN {X 0,Y 227.953,Z 376.717,A -85,B 0,C 180,E1 -19822.343,E2 -19822.343} C_VEL
LIN {X 0,Y 227.942,Z 376.703,A -85,B 0,C 180,E1 -19826.602,E2 -19826.602} C_VEL
LIN {X 0,Y 227.93,Z 376.936,A -85,B 0,C 180,E1 -19828.361,E2 -19828.361} C_VEL
LIN {X 0,Y 228.661,Z 379.09,A -85,B 0,C 180,E1 -19829.457,E2 -19829.457} C_VEL
LIN {X 0,Y 230.842,Z 382.02,A -85,B 0,C 180,E1 -19831.169,E2 -19831.169} C_VEL
LIN {X 0,Y 231.748,Z 384.142,A -85,B 0,C 180,E1 -19832.052,E2 -19832.052} C_VEL
LIN {X 0,Y 233.489,Z 386.608,A -85,B 0,C 180,E1 -19833.32,E2 -19833.32} C_VEL
LIN {X 0,Y 237.349,Z 393.238,A -85,B 0,C 180,E1 -19836.051,E2 -19836.051} C_VEL
LIN {X 0,Y 245.727,Z 404.556,A -85,B 0,C 180,E1 -19839.186,E2 -19839.186} C_VEL
LIN {X 0,Y 255.327,Z 418.832,A -85,B 0,C 180,E1 -19842.361,E2 -19842.361} C_VEL
LIN {X 0,Y 258.083,Z 423.787,A -85,B 0,C 180,E1 -19843.229,E2 -19843.229} C_VEL
LIN {X 0,Y 265.97,Z 442.833,A -85,B 0,C 180,E1 -19845.724,E2 -19845.724} C_VEL
LIN {X 0,Y 269.595,Z 452.266,A -85,B 0,C 180,E1 -19846.814,E2 -19846.814} C_VEL
LIN {X 0,Y 263.596,Z 563.933,A -85,B 0,C 180,E1 -19849.655,E2 -19849.655} C_VEL
LIN {X 0,Y 262.038,Z 578.746,A -85,B 0,C 180,E1 -19850.246,E2 -19850.246} C_VEL
LIN {X 0,Y 259.724,Z 593.971,A -85,B 0,C 180,E1 -19851.139,E2 -19851.139} C_VEL
LIN {X 0,Y 256.99,Z 608.07,A -85,B 0,C 180,E1 -19852.273,E2 -19852.273} C_VEL
LIN {X 0,Y 253.922,Z 621.622,A -85,B 0,C 180,E1 -19853.701,E2 -19853.701} C_VEL
LIN {X 0,Y 250.421,Z 634.382,A -85,B 0,C 180,E1 -19855.368,E2 -19855.368} C_VEL
LIN {X 0,Y 246.807,Z 646.032,A -85,B 0,C 180,E1 -19857.246,E2 -19857.246} C_VEL
LIN {X 0,Y 242.868,Z 657.716,A -85,B 0,C 180,E1 -19859.575,E2 -19859.575} C_VEL
LIN {X 0,Y 239.388,Z 667.537,A -85,B 0,C 180,E1 -19861.983,E2 -19861.983} C_VEL
LIN {X 0,Y 235.819,Z 677.13,A -85,B 0,C 180,E1 -19864.869,E2 -19864.869} C_VEL
LIN {X 0,Y 232.785,Z 685.109,A -85,B 0,C 180,E1 -19867.828,E2 -19867.828} C_VEL
LIN {X 0,Y 229.915,Z 692.697,A -85,B 0,C 180,E1 -19871.37,E2 -19871.37} C_VEL
LIN {X 0,Y 228.023,Z 698.431,A -85,B 0,C 180,E1 -19874.812,E2 -19874.812} C_VEL
LIN {X 0,Y 226.895,Z 701.908,A -85,B 0,C 180,E1 -19877.478,E2 -19877.478} C_VEL
LIN {X 0,Y 226.022,Z 705.433,A -85,B 0,C 180,E1 -19881.056,E2 -19881.056} C_VEL
LIN {X 0,Y 225.641,Z 707.75,A -85,B 0,C 180,E1 -19884.639,E2 -19884.639} C_VEL
LIN {X 0,Y 225.576,Z 708.913,A -85,B 0,C 180,E1 -19888.215,E2 -19888.215} C_VEL
LIN {X 0,Y 225.576,Z 708.911,A -85,B 0,C 180,E1 -19891.786,E2 -19891.786} C_VEL
LIN {X 0,Y 225.641,Z 707.736,A -85,B 0,C 180,E1 -19895.362,E2 -19895.362} C_VEL
LIN {X 0,Y 226.022,Z 705.404,A -85,B 0,C 180,E1 -19898.944,E2 -19898.944} C_VEL
LIN {X 0,Y 226.898,Z 701.857,A -85,B 0,C 180,E1 -19902.523,E2 -19902.523} C_VEL
LIN {X 0,Y 228.454,Z 697.013,A -85,B 0,C 180,E1 -19906.074,E2 -19906.074} C_VEL
LIN {X 0,Y 230.637,Z 690.748,A -85,B 0,C 180,E1 -19909.585,E2 -19909.585} C_VEL
LIN {X 0,Y 231.851,Z 687.676,A -85,B 0,C 180,E1 -19911.098,E2 -19911.098} C_VEL
LIN {X 0,Y 235.802,Z 682.846,A -85,B 0,C 180,E1 -19914.662,E2 -19914.662} C_VEL
LIN {X 0,Y 240.492,Z 677.15,A -85,B 0,C 180,E1 -19917.877,E2 -19917.877} C_VEL
LIN {X 0,Y 246.104,Z 670.212,A -85,B 0,C 180,E1 -19920.933,E2 -19920.933} C_VEL
LIN {X 0,Y 252.649,Z 661.915,A -85,B 0,C 180,E1 -19923.804,E2 -19923.804} C_VEL
LIN {X 0,Y 260.01,Z 652.109,A -85,B 0,C 180,E1 -19926.488,E2 -19926.488} C_VEL
LIN {X 0,Y 268.214,Z 640.543,A -85,B 0,C 180,E1 -19928.967,E2 -19928.967} C_VEL
LIN {X 0,Y 276.056,Z 628.688,A -85,B 0,C 180,E1 -19930.962,E2 -19930.962} C_VEL
LIN {X 0,Y 283.879,Z 615.911,A -85,B 0,C 180,E1 -19932.666,E2 -19932.666} C_VEL
LIN {X 0,Y 291.623,Z 601.986,A -85,B 0,C 180,E1 -19934.097,E2 -19934.097} C_VEL
LIN {X 0,Y 298.58,Z 587.974,A -85,B 0,C 180,E1 -19935.185,E2 -19935.185} C_VEL
LIN {X 0,Y 305.079,Z 572.868,A -85,B 0,C 180,E1 -19936.094,E2 -19936.094} C_VEL
LIN {X 0,Y 307.496,Z 566.606,A -85,B 0,C 180,E1 -19936.388,E2 -19936.388} C_VEL
LIN {X 0,Y 307.442,Z 566.645,A -85,B 0,C 180,E1 -19936.703,E2 -19936.703} C_VEL
LIN {X 0,Y 301.921,Z 580.035,A -85,B 0,C 180,E1 -19937.542,E2 -19937.542} C_VEL
LIN {X 0,Y 295.939,Z 592.573,A -85,B 0,C 180,E1 -19938.549,E2 -19938.549} C_VEL
LIN {X 0,Y 288.383,Z 606.512,A -85,B 0,C 180,E1 -19940.002,E2 -19940.002} C_VEL
LIN {X 0,Y 281.777,Z 617.455,A -85,B 0,C 180,E1 -19941.425,E2 -19941.425} C_VEL
LIN {X 0,Y 273.877,Z 629.35,A -85,B 0,C 180,E1 -19943.372,E2 -19943.372} C_VEL
LIN {X 0,Y 266.524,Z 639.478,A -85,B 0,C 180,E1 -19945.463,E2 -19945.463} C_VEL
LIN {X 0,Y 258.954,Z 649.188,A -85,B 0,C 180,E1 -19948.047,E2 -19948.047} C_VEL
LIN {X 0,Y 252.107,Z 657.22,A -85,B 0,C 180,E1 -19950.801,E2 -19950.801} C_VEL
LIN {X 0,Y 245.946,Z 663.8,A -85,B 0,C 180,E1 -19953.71,E2 -19953.71} C_VEL
LIN {X 0,Y 240.571,Z 668.99,A -85,B 0,C 180,E1 -19956.772,E2 -19956.772} C_VEL
LIN {X 0,Y 237.191,Z 671.982,A -85,B 0,C 180,E1 -19959.172,E2 -19959.172} C_VEL
LIN {X 0,Y 233.373,Z 674.888,A -85,B 0,C 180,E1 -19962.474,E2 -19962.474} C_VEL
LIN {X 0,Y 230.52,Z 676.543,A -85,B 0,C 180,E1 -19965.883,E2 -19965.883} C_VEL
LIN {X 0,Y 228.298,Z 676.981,A -85,B 0,C 180,E1 -19969.356,E2 -19969.356} C_VEL
LIN {X 0,Y 226.837,Z 676.148,A -85,B 0,C 180,E1 -19972.881,E2 -19972.881} C_VEL
LIN {X 0,Y 226.162,Z 674.012,A -85,B 0,C 180,E1 -19976.437,E2 -19976.437} C_VEL
LIN {X 0,Y 225.883,Z 670.505,A -85,B 0,C 180,E1 -19980,E2 -19980} C_VEL
LIN {X 0,Y 225.844,Z 666.913,A -85,B 0,C 180,E1 -19982.676,E2 -19982.676} C_VEL
LIN {X 0,Y 226.048,Z 660.814,A -85,B 0,C 180,E1 -19986.158,E2 -19986.158} C_VEL
LIN {X 0,Y 226.515,Z 653.624,A -85,B 0,C 180,E1 -19989.375,E2 -19989.375} C_VEL
LIN {X 0,Y 227.314,Z 644.955,A -85,B 0,C 180,E1 -19992.499,E2 -19992.499} C_VEL
LIN {X 0,Y 228.37,Z 635.994,A -85,B 0,C 180,E1 -19995.164,E2 -19995.164} C_VEL
LIN {X 0,Y 229.621,Z 625.282,A -85,B 0,C 180,E1 -19997.823,E2 -19997.823} C_VEL
LIN {X 0,Y 231.205,Z 613.539,A -85,B 0,C 180,E1 -20000.229,E2 -20000.229} C_VEL
LIN {X 0,Y 232.812,Z 600.675,A -85,B 0,C 180,E1 -20002.403,E2 -20002.403} C_VEL
LIN {X 0,Y 234.69,Z 586.809,A -85,B 0,C 180,E1 -20004.315,E2 -20004.315} C_VEL
LIN {X 0,Y 236.267,Z 572.522,A -85,B 0,C 180,E1 -20005.906,E2 -20005.906} C_VEL
LIN {X 0,Y 237.744,Z 556.98,A -85,B 0,C 180,E1 -20007.244,E2 -20007.244} C_VEL
LIN {X 0,Y 239.054,Z 540.18,A -85,B 0,C 180,E1 -20008.299,E2 -20008.299} C_VEL
LIN {X 0,Y 245.554,Z 446.258,A -85,B 0,C 180,E1 -20012.792,E2 -20012.792} C_VEL
LIN {X 0,Y 243.151,Z 427.313,A -85,B 0,C 180,E1 -20013.985,E2 -20013.985} C_VEL
LIN {X 0,Y 236.499,Z 408.004,A -85,B 0,C 180,E1 -20015.66,E2 -20015.66} C_VEL
LIN {X 0,Y 236.283,Z 406.443,A -85,B 0,C 180,E1 -20016.009,E2 -20016.009} C_VEL
LIN {X 0,Y 236.939,Z 405.78,A -85,B 0,C 180,E1 -20016.387,E2 -20016.387} C_VEL
LIN {X 0,Y 238.607,Z 404.498,A -85,B 0,C 180,E1 -20016.887,E2 -20016.887} C_VEL
LIN {X 0,Y 238.969,Z 404.068,A -85,B 0,C 180,E1 -20016.981,E2 -20016.981} C_VEL
LIN {X 0,Y 241.501,Z 405.011,A -85,B 0,C 180,E1 -20017.813,E2 -20017.813} C_VEL
LIN {X 0,Y 244.807,Z 407.348,A -85,B 0,C 180,E1 -20018.903,E2 -20018.903} C_VEL
LIN {X 0,Y 251.538,Z 418.261,A -85,B 0,C 180,E1 -20021.223,E2 -20021.223} C_VEL
LIN {X 0,Y 257.912,Z 429.671,A -85,B 0,C 180,E1 -20023.265,E2 -20023.265} C_VEL
LIN {X 0,Y 263.69,Z 441.337,A -85,B 0,C 180,E1 -20025.019,E2 -20025.019} C_VEL
LIN {X 0,Y 269.328,Z 454.282,A -85,B 0,C 180,E1 -20026.668,E2 -20026.668} C_VEL
LIN {X 0,Y 269.785,Z 456.464,A -85,B 0,C 180,E1 -20026.837,E2 -20026.837} C_VEL
LIN {X 0,Y 265.527,Z 537.349,A -85,B 0,C 180,E1 -20028.885,E2 -20028.885} C_VEL
LIN {X 0,Y 263.747,Z 567.143,A -85,B 0,C 180,E1 -20029.683,E2 -20029.683} C_VEL
LIN {X 0,Y 261.956,Z 582.518,A -85,B 0,C 180,E1 -20030.355,E2 -20030.355} C_VEL
LIN {X 0,Y 259.432,Z 597.916,A -85,B 0,C 180,E1 -20031.335,E2 -20031.335} C_VEL
LIN {X 0,Y 256.661,Z 611.635,A -85,B 0,C 180,E1 -20032.514,E2 -20032.514} C_VEL
LIN {X 0,Y 253.201,Z 626.042,A -85,B 0,C 180,E1 -20034.125,E2 -20034.125} C_VEL
LIN {X 0,Y 249.419,Z 639.063,A -85,B 0,C 180,E1 -20035.942,E2 -20035.942} C_VEL
LIN {X 0,Y 245.603,Z 651.068,A -85,B 0,C 180,E1 -20038.036,E2 -20038.036} C_VEL
LIN {X 0,Y 241.759,Z 662.037,A -85,B 0,C 180,E1 -20040.383,E2 -20040.383} C_VEL
LIN {X 0,Y 238.532,Z 671.273,A -85,B 0,C 180,E1 -20042.826,E2 -20042.826} C_VEL
LIN {X 0,Y 234.962,Z 680.35,A -85,B 0,C 180,E1 -20045.715,E2 -20045.715} C_VEL
LIN {X 0,Y 232.104,Z 687.887,A -85,B 0,C 180,E1 -20048.693,E2 -20048.693} C_VEL
LIN {X 0,Y 229.535,Z 694.916,A -85,B 0,C 180,E1 -20052.17,E2 -20052.17} C_VEL
LIN {X 0,Y 227.661,Z 700.444,A -85,B 0,C 180,E1 -20055.702,E2 -20055.702} C_VEL
LIN {X 0,Y 226.442,Z 704.628,A -85,B 0,C 180,E1 -20059.267,E2 -20059.267} C_VEL
LIN {X 0,Y 225.764,Z 707.566,A -85,B 0,C 180,E1 -20062.847,E2 -20062.847} C_VEL
LIN {X 0,Y 225.523,Z 709.326,A -85,B 0,C 180,E1 -20066.426,E2 -20066.426} C_VEL
LIN {X 0,Y 225.586,Z 709.934,A -85,B 0,C 180,E1 -20070,E2 -20070} C_VEL
LIN {X 0,Y 225.524,Z 709.358,A -85,B 0,C 180,E1 -20073.573,E2 -20073.573} C_VEL
LIN {X 0,Y 225.764,Z 707.643,A -85,B 0,C 180,E1 -20077.153,E2 -20077.153} C_VEL
LIN {X 0,Y 226.435,Z 704.755,A -85,B 0,C 180,E1 -20080.732,E2 -20080.732} C_VEL
LIN {X 0,Y 227.635,Z 700.627,A -85,B 0,C 180,E1 -20084.299,E2 -20084.299} C_VEL
LIN {X 0,Y 229.496,Z 695.147,A -85,B 0,C 180,E1 -20087.832,E2 -20087.832} C_VEL
LIN {X 0,Y 232.028,Z 688.168,A -85,B 0,C 180,E1 -20091.313,E2 -20091.313} C_VEL
LIN {X 0,Y 234.871,Z 680.696,A -85,B 0,C 180,E1 -20094.295,E2 -20094.295} C_VEL
LIN {X 0,Y 238.424,Z 671.694,A -85,B 0,C 180,E1 -20097.187,E2 -20097.187} C_VEL
LIN {X 0,Y 241.653,Z 662.496,A -85,B 0,C 180,E1 -20099.631,E2 -20099.631} C_VEL
LIN {X 0,Y 245.847,Z 650.655,A -85,B 0,C 180,E1 -20102.17,E2 -20102.17} C_VEL
LIN {X 0,Y 249.676,Z 638.571,A -85,B 0,C 180,E1 -20104.261,E2 -20104.261} C_VEL
LIN {X 0,Y 253.371,Z 625.824,A -85,B 0,C 180,E1 -20106.024,E2 -20106.024} C_VEL
LIN {X 0,Y 256.619,Z 612.265,A -85,B 0,C 180,E1 -20107.543,E2 -20107.543} C_VEL
LIN {X 0,Y 259.489,Z 598.065,A -85,B 0,C 180,E1 -20108.779,E2 -20108.779} C_VEL
LIN {X 0,Y 262.039,Z 582.729,A -85,B 0,C 180,E1 -20109.754,E2 -20109.754} C_VEL
LIN {X 0,Y 263.827,Z 567.446,A -85,B 0,C 180,E1 -20110.427,E2 -20110.427} C_VEL
LIN {X 0,Y 265.48,Z 539.568,A -85,B 0,C 180,E1 -20111.186,E2 -20111.186} C_VEL
LIN {X 0,Y 269.952,Z 456.54,A -85,B 0,C 180,E1 -20113.268,E2 -20113.268} C_VEL
LIN {X 0,Y 269.493,Z 454.417,A -85,B 0,C 180,E1 -20113.436,E2 -20113.436} C_VEL
LIN {X 0,Y 263.042,Z 439.738,A -85,B 0,C 180,E1 -20115.33,E2 -20115.33} C_VEL
LIN {X 0,Y 255.3,Z 424.61,A -85,B 0,C 180,E1 -20117.721,E2 -20117.721} C_VEL
LIN {X 0,Y 246.92,Z 410.558,A -85,B 0,C 180,E1 -20120.518,E2 -20120.518} C_VEL
LIN {X 0,Y 239.921,Z 399.986,A -85,B 0,C 180,E1 -20123.094,E2 -20123.094} C_VEL
LIN {X 0,Y 236.405,Z 394.774,A -85,B 0,C 180,E1 -20124.574,E2 -20124.574} C_VEL
LIN {X 0,Y 233.79,Z 388.766,A -85,B 0,C 180,E1 -20127.321,E2 -20127.321} C_VEL
LIN {X 0,Y 229.72,Z 380.669,A -85,B 0,C 180,E1 -20131.692,E2 -20131.692} C_VEL
LIN {X 0,Y 228.068,Z 377.541,A -85,B 0,C 180,E1 -20133.611,E2 -20133.611} C_VEL
LIN {X 0,Y 227.94,Z 376.875,A -85,B 0,C 180,E1 -20134.092,E2 -20134.092} C_VEL
LIN {X 0,Y 227.085,Z 376.82,A -85,B 0,C 180,E1 -20135.552,E2 -20135.552} C_VEL
LIN {X 0,Y 224.213,Z 377.155,A -85,B 0,C 180,E1 -20137.96,E2 -20137.96} C_VEL
LIN {X 0,Y 221.908,Z 377.527,A -85,B 0,C 180,E1 -20139.934,E2 -20139.934} C_VEL
LIN {X 0,Y 220.96,Z 377.576,A -85,B 0,C 180,E1 -20141.465,E2 -20141.465} C_VEL
LIN {X 0,Y 220.898,Z 377.571,A -85,B 0,C 180,E1 -20141.983,E2 -20141.983} C_VEL
LIN {X 0,Y 220.969,Z 377.573,A -85,B 0,C 180,E1 -20145.259,E2 -20145.259} C_VEL
LIN {X 0,Y 221.202,Z 377.538,A -85,B 0,C 180,E1 -20150.859,E2 -20150.859} C_VEL
LIN {X 0,Y 221.254,Z 377.542,A -85,B 0,C 180,E1 -20152.7,E2 -20152.7} C_VEL
LIN {X 0,Y 221.507,Z 377.519,A -85,B 0,C 180,E1 -20158.182,E2 -20158.182} C_VEL
LIN {X 0,Y 221.51,Z 377.484,A -85,B 0,C 180,E1 -20161.818,E2 -20161.818} C_VEL
LIN {X 0,Y 221.241,Z 377.517,A -85,B 0,C 180,E1 -20167.3,E2 -20167.3} C_VEL
LIN {X 0,Y 221.063,Z 377.571,A -85,B 0,C 180,E1 -20170.996,E2 -20170.996} C_VEL
LIN {X 0,Y 220.986,Z 377.582,A -85,B 0,C 180,E1 -20176.632,E2 -20176.632} C_VEL
LIN {X 0,Y 220.893,Z 377.568,A -85,B 0,C 180,E1 -20180.486,E2 -20180.486} C_VEL
LIN {X 0,Y 220.871,Z 377.73,A -85,B 0,C 180,E1 -20184.685,E2 -20184.685} C_VEL
LIN {X 0,Y 221.088,Z 378.554,A -85,B 0,C 180,E1 -20185.413,E2 -20185.413} C_VEL
LIN {X 0,Y 222.749,Z 381.595,A -85,B 0,C 180,E1 -20187.273,E2 -20187.273} C_VEL
LIN {X 0,Y 223.781,Z 382.645,A -85,B 0,C 180,E1 -20188.105,E2 -20188.105} C_VEL
LIN {X 0,Y 224.53,Z 384.601,A -85,B 0,C 180,E1 -20189.022,E2 -20189.022} C_VEL
LIN {X 0,Y 226.652,Z 387.569,A -85,B 0,C 180,E1 -20190.772,E2 -20190.772} C_VEL
LIN {X 0,Y 227.552,Z 389.641,A -85,B 0,C 180,E1 -20191.671,E2 -20191.671} C_VEL
LIN {X 0,Y 229.27,Z 392.18,A -85,B 0,C 180,E1 -20192.98,E2 -20192.98} C_VEL
LIN {X 0,Y 232.752,Z 396.89,A -85,B 0,C 180,E1 -20194.653,E2 -20194.653} C_VEL
LIN {X 0,Y 239.792,Z 406.321,A -85,B 0,C 180,E1 -20197.488,E2 -20197.488} C_VEL
LIN {X 0,Y 247.212,Z 417.194,A -85,B 0,C 180,E1 -20200.17,E2 -20200.17} C_VEL
LIN {X 0,Y 253.492,Z 427.174,A -85,B 0,C 180,E1 -20202.247,E2 -20202.247} C_VEL
LIN {X 0,Y 261.297,Z 446.334,A -85,B 0,C 180,E1 -20204.845,E2 -20204.845} C_VEL
LIN {X 0,Y 264.341,Z 454.404,A -85,B 0,C 180,E1 -20205.808,E2 -20205.808} C_VEL
LIN {X 0,Y 258.236,Z 564.048,A -85,B 0,C 180,E1 -20208.637,E2 -20208.637} C_VEL
LIN {X 0,Y 256.627,Z 578.817,A -85,B 0,C 180,E1 -20209.233,E2 -20209.233} C_VEL
LIN {X 0,Y 254.232,Z 594.023,A -85,B 0,C 180,E1 -20210.134,E2 -20210.134} C_VEL
LIN {X 0,Y 251.402,Z 608.111,A -85,B 0,C 180,E1 -20211.281,E2 -20211.281} C_VEL
LIN {X 0,Y 248.141,Z 621.998,A -85,B 0,C 180,E1 -20212.77,E2 -20212.77} C_VEL
LIN {X 0,Y 244.598,Z 634.412,A -85,B 0,C 180,E1 -20214.42,E2 -20214.42} C_VEL
LIN {X 0,Y 240.838,Z 646.058,A -85,B 0,C 180,E1 -20216.328,E2 -20216.328} C_VEL
LIN {X 0,Y 236.736,Z 657.739,A -85,B 0,C 180,E1 -20218.7,E2 -20218.7} C_VEL
LIN {X 0,Y 233.058,Z 667.558,A -85,B 0,C 180,E1 -20221.152,E2 -20221.152} C_VEL
LIN {X 0,Y 229.891,Z 675.923,A -85,B 0,C 180,E1 -20223.687,E2 -20223.687} C_VEL
LIN {X 0,Y 226.571,Z 684.092,A -85,B 0,C 180,E1 -20226.704,E2 -20226.704} C_VEL
LIN {X 0,Y 223.894,Z 690.846,A -85,B 0,C 180,E1 -20229.801,E2 -20229.801} C_VEL
LIN {X 0,Y 221.566,Z 697.099,A -85,B 0,C 180,E1 -20233.413,E2 -20233.413} C_VEL
LIN {X 0,Y 219.916,Z 701.923,A -85,B 0,C 180,E1 -20237.074,E2 -20237.074} C_VEL
LIN {X 0,Y 218.983,Z 705.447,A -85,B 0,C 180,E1 -20240.766,E2 -20240.766} C_VEL
LIN {X 0,Y 218.562,Z 707.764,A -85,B 0,C 180,E1 -20244.464,E2 -20244.464} C_VEL
LIN {X 0,Y 218.478,Z 708.927,A -85,B 0,C 180,E1 -20248.157,E2 -20248.157} C_VEL
LIN {X 0,Y 218.479,Z 708.924,A -85,B 0,C 180,E1 -20251.844,E2 -20251.844} C_VEL
LIN {X 0,Y 218.563,Z 707.75,A -85,B 0,C 180,E1 -20255.536,E2 -20255.536} C_VEL
LIN {X 0,Y 218.984,Z 705.417,A -85,B 0,C 180,E1 -20259.234,E2 -20259.234} C_VEL
LIN {X 0,Y 219.919,Z 701.87,A -85,B 0,C 180,E1 -20262.927,E2 -20262.927} C_VEL
LIN {X 0,Y 221.567,Z 697.027,A -85,B 0,C 180,E1 -20266.588,E2 -20266.588} C_VEL
LIN {X 0,Y 223.914,Z 690.768,A -85,B 0,C 180,E1 -20270.198,E2 -20270.198} C_VEL
LIN {X 0,Y 225.011,Z 688.293,A -85,B 0,C 180,E1 -20271.531,E2 -20271.531} C_VEL
LIN {X 0,Y 229.404,Z 683.612,A -85,B 0,C 180,E1 -20275.398,E2 -20275.398} C_VEL
LIN {X 0,Y 234.315,Z 678.256,A -85,B 0,C 180,E1 -20278.679,E2 -20278.679} C_VEL
LIN {X 0,Y 240.181,Z 671.724,A -85,B 0,C 180,E1 -20281.783,E2 -20281.783} C_VEL
LIN {X 0,Y 247.924,Z 662.856,A -85,B 0,C 180,E1 -20285.032,E2 -20285.032} C_VEL
LIN {X 0,Y 255.661,Z 653.464,A -85,B 0,C 180,E1 -20287.709,E2 -20287.709} C_VEL
LIN {X 0,Y 264.246,Z 642.447,A -85,B 0,C 180,E1 -20290.163,E2 -20290.163} C_VEL
LIN {X 0,Y 272.414,Z 631.177,A -85,B 0,C 180,E1 -20292.127,E2 -20292.127} C_VEL
LIN {X 0,Y 281.147,Z 618.051,A -85,B 0,C 180,E1 -20293.923,E2 -20293.923} C_VEL
LIN {X 0,Y 289.856,Z 603.556,A -85,B 0,C 180,E1 -20295.419,E2 -20295.419} C_VEL
LIN {X 0,Y 297.439,Z 589.349,A -85,B 0,C 180,E1 -20296.503,E2 -20296.503} C_VEL
LIN {X 0,Y 297.576,Z 588.998,A -85,B 0,C 180,E1 -20296.772,E2 -20296.772} C_VEL
LIN {X 0,Y 290.21,Z 602.34,A -85,B 0,C 180,E1 -20298.011,E2 -20298.011} C_VEL
LIN {X 0,Y 281.869,Z 615.698,A -85,B 0,C 180,E1 -20299.589,E2 -20299.589} C_VEL
LIN {X 0,Y 273.432,Z 627.8,A -85,B 0,C 180,E1 -20301.443,E2 -20301.443} C_VEL
LIN {X 0,Y 264.43,Z 639.408,A -85,B 0,C 180,E1 -20303.747,E2 -20303.747} C_VEL
LIN {X 0,Y 256.296,Z 649.055,A -85,B 0,C 180,E1 -20306.27,E2 -20306.27} C_VEL
LIN {X 0,Y 249.758,Z 656.184,A -85,B 0,C 180,E1 -20308.629,E2 -20308.629} C_VEL
LIN {X 0,Y 243.013,Z 662.955,A -85,B 0,C 180,E1 -20311.499,E2 -20311.499} C_VEL
LIN {X 0,Y 236.882,Z 668.434,A -85,B 0,C 180,E1 -20314.52,E2 -20314.52} C_VEL
LIN {X 0,Y 233.025,Z 671.63,A -85,B 0,C 180,E1 -20316.916,E2 -20316.916} C_VEL
LIN {X 0,Y 228.541,Z 674.818,A -85,B 0,C 180,E1 -20320.229,E2 -20320.229} C_VEL
LIN {X 0,Y 225.071,Z 676.769,A -85,B 0,C 180,E1 -20323.678,E2 -20323.678} C_VEL
LIN {X 0,Y 222.423,Z 677.516,A -85,B 0,C 180,E1 -20327.222,E2 -20327.222} C_VEL
LIN {X 0,Y 220.498,Z 677.031,A -85,B 0,C 180,E1 -20330.83,E2 -20330.83} C_VEL
LIN {X 0,Y 219.349,Z 675.279,A -85,B 0,C 180,E1 -20334.484,E2 -20334.484} C_VEL
LIN {X 0,Y 218.928,Z 672.215,A -85,B 0,C 180,E1 -20338.161,E2 -20338.161} C_VEL
LIN {X 0,Y 218.768,Z 667.713,A -85,B 0,C 180,E1 -20341.841,E2 -20341.841} C_VEL
LIN {X 0,Y 218.814,Z 662.601,A -85,B 0,C 180,E1 -20344.975,E2 -20344.975} C_VEL
LIN {X 0,Y 219.256,Z 655.817,A -85,B 0,C 180,E1 -20348.294,E2 -20348.294} C_VEL
LIN {X 0,Y 219.922,Z 647.555,A -85,B 0,C 180,E1 -20351.521,E2 -20351.521} C_VEL
LIN {X 0,Y 220.837,Z 639.03,A -85,B 0,C 180,E1 -20354.279,E2 -20354.279} C_VEL
LIN {X 0,Y 222.11,Z 628.853,A -85,B 0,C 180,E1 -20357.019,E2 -20357.019} C_VEL
LIN {X 0,Y 223.746,Z 616.466,A -85,B 0,C 180,E1 -20359.768,E2 -20359.768} C_VEL
LIN {X 0,Y 225.454,Z 603.086,A -85,B 0,C 180,E1 -20362.208,E2 -20362.208} C_VEL
LIN {X 0,Y 227.297,Z 589.683,A -85,B 0,C 180,E1 -20364.185,E2 -20364.185} C_VEL
LIN {X 0,Y 229.133,Z 573.939,A -85,B 0,C 180,E1 -20366.04,E2 -20366.04} C_VEL
LIN {X 0,Y 230.538,Z 559.558,A -85,B 0,C 180,E1 -20367.37,E2 -20367.37} C_VEL
LIN {X 0,Y 231.895,Z 543.478,A -85,B 0,C 180,E1 -20368.478,E2 -20368.478} C_VEL
LIN {X 0,Y 238.794,Z 447.018,A -85,B 0,C 180,E1 -20373.287,E2 -20373.287} C_VEL
LIN {X 0,Y 236.586,Z 429.425,A -85,B 0,C 180,E1 -20374.433,E2 -20374.433} C_VEL
LIN {X 0,Y 233.434,Z 419.974,A -85,B 0,C 180,E1 -20375.29,E2 -20375.29} C_VEL
LIN {X 0,Y 233.308,Z 418.368,A -85,B 0,C 180,E1 -20375.683,E2 -20375.683} C_VEL
LIN {X 0,Y 234.987,Z 417.308,A -85,B 0,C 180,E1 -20376.351,E2 -20376.351} C_VEL
LIN {X 0,Y 236.763,Z 414.904,A -85,B 0,C 180,E1 -20376.81,E2 -20376.81} C_VEL
LIN {X 0,Y 238.183,Z 412.162,A -85,B 0,C 180,E1 -20377.128,E2 -20377.128} C_VEL
LIN {X 0,Y 238.859,Z 411.763,A -85,B 0,C 180,E1 -20377.321,E2 -20377.321} C_VEL
LIN {X 0,Y 240.097,Z 412.087,A -85,B 0,C 180,E1 -20377.721,E2 -20377.721} C_VEL
LIN {X 0,Y 241.96,Z 413.613,A -85,B 0,C 180,E1 -20378.357,E2 -20378.357} C_VEL
LIN {X 0,Y 248.167,Z 423.887,A -85,B 0,C 180,E1 -20380.576,E2 -20380.576} C_VEL
LIN {X 0,Y 254.162,Z 434.911,A -85,B 0,C 180,E1 -20382.577,E2 -20382.577} C_VEL
LIN {X 0,Y 260.346,Z 447.682,A -85,B 0,C 180,E1 -20384.527,E2 -20384.527} C_VEL
LIN {X 0,Y 264.578,Z 457.806,A -85,B 0,C 180,E1 -20385.824,E2 -20385.824} C_VEL
LIN {X 0,Y 259.832,Z 544.39,A -85,B 0,C 180,E1 -20388.041,E2 -20388.041} C_VEL
LIN {X 0,Y 258.38,Z 567.073,A -85,B 0,C 180,E1 -20388.665,E2 -20388.665} C_VEL
LIN {X 0,Y 256.515,Z 582.473,A -85,B 0,C 180,E1 -20389.34,E2 -20389.34} C_VEL
LIN {X 0,Y 253.922,Z 597.883,A -85,B 0,C 180,E1 -20390.333,E2 -20390.333} C_VEL
LIN {X 0,Y 251.074,Z 611.608,A -85,B 0,C 180,E1 -20391.529,E2 -20391.529} C_VEL
LIN {X 0,Y 247.789,Z 624.921,A -85,B 0,C 180,E1 -20393.022,E2 -20393.022} C_VEL
LIN {X 0,Y 243.921,Z 637.848,A -85,B 0,C 180,E1 -20394.812,E2 -20394.812} C_VEL
LIN {X 0,Y 239.903,Z 650.05,A -85,B 0,C 180,E1 -20396.932,E2 -20396.932} C_VEL
LIN {X 0,Y 235.576,Z 662.021,A -85,B 0,C 180,E1 -20399.524,E2 -20399.524} C_VEL
LIN {X 0,Y 232.193,Z 671.258,A -85,B 0,C 180,E1 -20402.02,E2 -20402.02} C_VEL
LIN {X 0,Y 228.462,Z 680.335,A -85,B 0,C 180,E1 -20404.977,E2 -20404.977} C_VEL
LIN {X 0,Y 225.442,Z 687.873,A -85,B 0,C 180,E1 -20408.032,E2 -20408.032} C_VEL
LIN {X 0,Y 222.715,Z 694.902,A -85,B 0,C 180,E1 -20411.605,E2 -20411.605} C_VEL
LIN {X 0,Y 220.757,Z 700.431,A -85,B 0,C 180,E1 -20415.245,E2 -20415.245} C_VEL
LIN {X 0,Y 219.411,Z 704.614,A -85,B 0,C 180,E1 -20418.919,E2 -20418.919} C_VEL
LIN {X 0,Y 218.685,Z 707.553,A -85,B 0,C 180,E1 -20422.614,E2 -20422.614} C_VEL
LIN {X 0,Y 218.43,Z 709.312,A -85,B 0,C 180,E1 -20426.31,E2 -20426.31} C_VEL
LIN {X 0,Y 218.487,Z 709.921,A -85,B 0,C 180,E1 -20430,E2 -20430} C_VEL
LIN {X 0,Y 218.45,Z 709.344,A -85,B 0,C 180,E1 -20433.689,E2 -20433.689} C_VEL
LIN {X 0,Y 218.685,Z 707.628,A -85,B 0,C 180,E1 -20437.386,E2 -20437.386} C_VEL
LIN {X 0,Y 219.402,Z 704.74,A -85,B 0,C 180,E1 -20441.081,E2 -20441.081} C_VEL
LIN {X 0,Y 220.728,Z 700.611,A -85,B 0,C 180,E1 -20444.757,E2 -20444.757} C_VEL
LIN {X 0,Y 222.66,Z 695.13,A -85,B 0,C 180,E1 -20448.399,E2 -20448.399} C_VEL
LIN {X 0,Y 225.371,Z 688.151,A -85,B 0,C 180,E1 -20451.975,E2 -20451.975} C_VEL
LIN {X 0,Y 228.352,Z 680.677,A -85,B 0,C 180,E1 -20455.036,E2 -20455.036} C_VEL
LIN {X 0,Y 232.086,Z 671.674,A -85,B 0,C 180,E1 -20457.993,E2 -20457.993} C_VEL
LIN {X 0,Y 235.479,Z 662.474,A -85,B 0,C 180,E1 -20460.489,E2 -20460.489} C_VEL
LIN {X 0,Y 239.814,Z 650.63,A -85,B 0,C 180,E1 -20463.081,E2 -20463.081} C_VEL
LIN {X 0,Y 243.826,Z 638.543,A -85,B 0,C 180,E1 -20465.203,E2 -20465.203} C_VEL
LIN {X 0,Y 247.892,Z 624.882,A -85,B 0,C 180,E1 -20467.108,E2 -20467.108} C_VEL
LIN {X 0,Y 251.035,Z 612.227,A -85,B 0,C 180,E1 -20468.529,E2 -20468.529} C_VEL
LIN {X 0,Y 253.995,Z 598.017,A -85,B 0,C 180,E1 -20469.781,E2 -20469.781} C_VEL
LIN {X 0,Y 256.622,Z 582.664,A -85,B 0,C 180,E1 -20470.768,E2 -20470.768} C_VEL
LIN {X 0,Y 258.469,Z 567.348,A -85,B 0,C 180,E1 -20471.447,E2 -20471.447} C_VEL
LIN {X 0,Y 260.301,Z 537.635,A -85,B 0,C 180,E1 -20472.257,E2 -20472.257} C_VEL
LIN {X 0,Y 264.742,Z 457.975,A -85,B 0,C 180,E1 -20474.28,E2 -20474.28} C_VEL
LIN {X 0,Y 258.686,Z 443.978,A -85,B 0,C 180,E1 -20476.142,E2 -20476.142} C_VEL
LIN {X 0,Y 252.324,Z 431.325,A -85,B 0,C 180,E1 -20478.184,E2 -20478.184} C_VEL
LIN {X 0,Y 247.506,Z 422.738,A -85,B 0,C 180,E1 -20479.816,E2 -20479.816} C_VEL
LIN {X 0,Y 240.91,Z 411.752,A -85,B 0,C 180,E1 -20482.22,E2 -20482.22} C_VEL
LIN {X 0,Y 235.381,Z 403.614,A -85,B 0,C 180,E1 -20484.396,E2 -20484.396} C_VEL
LIN {X 0,Y 230.886,Z 397.321,A -85,B 0,C 180,E1 -20486.319,E2 -20486.319} C_VEL
LIN {X 0,Y 229.15,Z 394.595,A -85,B 0,C 180,E1 -20487.22,E2 -20487.22} C_VEL
LIN {X 0,Y 226.167,Z 388.498,A -85,B 0,C 180,E1 -20490.468,E2 -20490.468} C_VEL
LIN {X 0,Y 223.366,Z 382.82,A -85,B 0,C 180,E1 -20493.864,E2 -20493.864} C_VEL
LIN {X 0,Y 220.975,Z 378.224,A -85,B 0,C 180,E1 -20497.064,E2 -20497.064} C_VEL
LIN {X 0,Y 220.907,Z 377.584,A -85,B 0,C 180,E1 -20498.049,E2 -20498.049} C_VEL
LIN {X 0,Y 220.898,Z 377.571,A -85,B 0,C 180,E1 -20501.983,E2 -20501.983} C_VEL
LIN {X 0,Y 220.287,Z 377.649,A -85,B 0,C 180,E1 -20503.505,E2 -20503.505} C_VEL
LIN {X 0,Y 217.535,Z 378.014,A -85,B 0,C 180,E1 -20505.992,E2 -20505.992} C_VEL
LIN {X 0,Y 215.185,Z 378.287,A -85,B 0,C 180,E1 -20508.023,E2 -20508.023} C_VEL
LIN {X 0,Y 214.196,Z 378.399,A -85,B 0,C 180,E1 -20509.597,E2 -20509.597} C_VEL
LIN {X 0,Y 214.126,Z 378.41,A -85,B 0,C 180,E1 -20510.13,E2 -20510.13} C_VEL
LIN {X 0,Y 214.194,Z 378.425,A -85,B 0,C 180,E1 -20512.458,E2 -20512.458} C_VEL
LIN {X 0,Y 214.44,Z 378.398,A -85,B 0,C 180,E1 -20518.122,E2 -20518.122} C_VEL
LIN {X 0,Y 214.546,Z 378.359,A -85,B 0,C 180,E1 -20520,E2 -20520} C_VEL
LIN {X 0,Y 214.443,Z 378.364,A -85,B 0,C 180,E1 -20521.878,E2 -20521.878} C_VEL
LIN {X 0,Y 214.183,Z 378.395,A -85,B 0,C 180,E1 -20527.542,E2 -20527.542} C_VEL
LIN {X 0,Y 213.994,Z 378.444,A -85,B 0,C 180,E1 -20531.364,E2 -20531.364} C_VEL
LIN {X 0,Y 213.904,Z 378.439,A -85,B 0,C 180,E1 -20535.239,E2 -20535.239} C_VEL
LIN {X 0,Y 213.826,Z 378.445,A -85,B 0,C 180,E1 -20539.188,E2 -20539.188} C_VEL
LIN {X 0,Y 213.9,Z 378.816,A -85,B 0,C 180,E1 -20540.683,E2 -20540.683} C_VEL
LIN {X 0,Y 215.293,Z 381.939,A -85,B 0,C 180,E1 -20543.062,E2 -20543.062} C_VEL
LIN {X 0,Y 217.142,Z 384.23,A -85,B 0,C 180,E1 -20545.009,E2 -20545.009} C_VEL
LIN {X 0,Y 218.591,Z 387.064,A -85,B 0,C 180,E1 -20546.751,E2 -20546.751} C_VEL
LIN {X 0,Y 219.627,Z 388.229,A -85,B 0,C 180,E1 -20547.645,E2 -20547.645} C_VEL
LIN {X 0,Y 221.416,Z 391.6,A -85,B 0,C 180,E1 -20549.471,E2 -20549.471} C_VEL
LIN {X 0,Y 222.769,Z 393.612,A -85,B 0,C 180,E1 -20550.513,E2 -20550.513} C_VEL
LIN {X 0,Y 225.263,Z 396.776,A -85,B 0,C 180,E1 -20551.768,E2 -20551.768} C_VEL
LIN {X 0,Y 233.123,Z 406.975,A -85,B 0,C 180,E1 -20555.317,E2 -20555.317} C_VEL
LIN {X 0,Y 240.616,Z 417.695,A -85,B 0,C 180,E1 -20558.286,E2 -20558.286} C_VEL
LIN {X 0,Y 249.308,Z 431.431,A -85,B 0,C 180,E1 -20561.353,E2 -20561.353} C_VEL
LIN {X 0,Y 256.316,Z 448.824,A -85,B 0,C 180,E1 -20563.807,E2 -20563.807} C_VEL
LIN {X 0,Y 259.196,Z 456.634,A -85,B 0,C 180,E1 -20564.772,E2 -20564.772} C_VEL
LIN {X 0,Y 252.955,Z 564.163,A -85,B 0,C 180,E1 -20567.576,E2 -20567.576} C_VEL
LIN {X 0,Y 251.292,Z 578.889,A -85,B 0,C 180,E1 -20568.176,E2 -20568.176} C_VEL
LIN {X 0,Y 248.833,Z 594.075,A -85,B 0,C 180,E1 -20569.088,E2 -20569.088} C_VEL
LIN {X 0,Y 245.899,Z 608.152,A -85,B 0,C 180,E1 -20570.246,E2 -20570.246} C_VEL
LIN {X 0,Y 242.849,Z 620.704,A -85,B 0,C 180,E1 -20571.591,E2 -20571.591} C_VEL
LIN {X 0,Y 238.855,Z 634.44,A -85,B 0,C 180,E1 -20573.428,E2 -20573.428} C_VEL
LIN {X 0,Y 234.922,Z 646.084,A -85,B 0,C 180,E1 -20575.361,E2 -20575.361} C_VEL
LIN {X 0,Y 230.675,Z 657.762,A -85,B 0,C 180,E1 -20577.78,E2 -20577.78} C_VEL
LIN {X 0,Y 226.782,Z 667.579,A -85,B 0,C 180,E1 -20580.275,E2 -20580.275} C_VEL
LIN {X 0,Y 223.525,Z 675.942,A -85,B 0,C 180,E1 -20582.877,E2 -20582.877} C_VEL
LIN {X 0,Y 220.028,Z 684.11,A -85,B 0,C 180,E1 -20585.968,E2 -20585.968} C_VEL
LIN {X 0,Y 217.2,Z 690.863,A -85,B 0,C 180,E1 -20589.15,E2 -20589.15} C_VEL
LIN {X 0,Y 214.705,Z 697.115,A -85,B 0,C 180,E1 -20592.867,E2 -20592.867} C_VEL
LIN {X 0,Y 212.954,Z 701.938,A -85,B 0,C 180,E1 -20596.643,E2 -20596.643} C_VEL
LIN {X 0,Y 211.96,Z 705.462,A -85,B 0,C 180,E1 -20600.457,E2 -20600.457} C_VEL
LIN {X 0,Y 211.483,Z 707.779,A -85,B 0,C 180,E1 -20604.279,E2 -20604.279} C_VEL
LIN {X 0,Y 211.384,Z 708.941,A -85,B 0,C 180,E1 -20608.095,E2 -20608.095} C_VEL
LIN {X 0,Y 211.385,Z 708.938,A -85,B 0,C 180,E1 -20611.906,E2 -20611.906} C_VEL
LIN {X 0,Y 211.483,Z 707.763,A -85,B 0,C 180,E1 -20615.722,E2 -20615.722} C_VEL
LIN {X 0,Y 211.96,Z 705.431,A -85,B 0,C 180,E1 -20619.543,E2 -20619.543} C_VEL
LIN {X 0,Y 212.958,Z 701.884,A -85,B 0,C 180,E1 -20623.357,E2 -20623.357} C_VEL
LIN {X 0,Y 214.705,Z 697.041,A -85,B 0,C 180,E1 -20627.134,E2 -20627.134} C_VEL
LIN {X 0,Y 217.216,Z 690.789,A -85,B 0,C 180,E1 -20630.849,E2 -20630.849} C_VEL
LIN {X 0,Y 217.937,Z 689.032,A -85,B 0,C 180,E1 -20631.768,E2 -20631.768} C_VEL
LIN {X 0,Y 223.03,Z 684.289,A -85,B 0,C 180,E1 -20636.178,E2 -20636.178} C_VEL
LIN {X 0,Y 228.185,Z 679.349,A -85,B 0,C 180,E1 -20639.525,E2 -20639.525} C_VEL
LIN {X 0,Y 234.319,Z 673.269,A -85,B 0,C 180,E1 -20642.676,E2 -20642.676} C_VEL
LIN {X 0,Y 242.371,Z 664.948,A -85,B 0,C 180,E1 -20645.958,E2 -20645.958} C_VEL
LIN {X 0,Y 250.393,Z 656.155,A -85,B 0,C 180,E1 -20648.647,E2 -20648.647} C_VEL
LIN {X 0,Y 259.254,Z 645.829,A -85,B 0,C 180,E1 -20651.101,E2 -20651.101} C_VEL
LIN {X 0,Y 268.884,Z 633.704,A -85,B 0,C 180,E1 -20653.324,E2 -20653.324} C_VEL
LIN {X 0,Y 277.936,Z 621.272,A -85,B 0,C 180,E1 -20655.074,E2 -20655.074} C_VEL
LIN {X 0,Y 286.987,Z 607.582,A -85,B 0,C 180,E1 -20656.536,E2 -20656.536} C_VEL
LIN {X 0,Y 287.751,Z 606.373,A -85,B 0,C 180,E1 -20656.655,E2 -20656.655} C_VEL
LIN {X 0,Y 287.858,Z 606.144,A -85,B 0,C 180,E1 -20656.873,E2 -20656.873} C_VEL
LIN {X 0,Y 279.835,Z 617.945,A -85,B 0,C 180,E1 -20658.276,E2 -20658.276} C_VEL
LIN {X 0,Y 271.016,Z 629.569,A -85,B 0,C 180,E1 -20660.073,E2 -20660.073} C_VEL
LIN {X 0,Y 262.722,Z 639.541,A -85,B 0,C 180,E1 -20662.029,E2 -20662.029} C_VEL
LIN {X 0,Y 255.03,Z 648.04,A -85,B 0,C 180,E1 -20664.155,E2 -20664.155} C_VEL
LIN {X 0,Y 247.916,Z 655.315,A -85,B 0,C 180,E1 -20666.441,E2 -20666.441} C_VEL
LIN {X 0,Y 240.509,Z 662.25,A -85,B 0,C 180,E1 -20669.245,E2 -20669.245} C_VEL
LIN {X 0,Y 233.82,Z 667.888,A -85,B 0,C 180,E1 -20672.232,E2 -20672.232} C_VEL
LIN {X 0,Y 229.313,Z 671.282,A -85,B 0,C 180,E1 -20674.592,E2 -20674.592} C_VEL
LIN {X 0,Y 224.241,Z 674.677,A -85,B 0,C 180,E1 -20677.908,E2 -20677.908} C_VEL
LIN {X 0,Y 220.029,Z 676.895,A -85,B 0,C 180,E1 -20681.373,E2 -20681.373} C_VEL
LIN {X 0,Y 216.861,Z 677.918,A -85,B 0,C 180,E1 -20684.974,E2 -20684.974} C_VEL
LIN {X 0,Y 214.388,Z 677.765,A -85,B 0,C 180,E1 -20688.657,E2 -20688.657} C_VEL
LIN {X 0,Y 212.775,Z 676.375,A -85,B 0,C 180,E1 -20692.408,E2 -20692.408} C_VEL
LIN {X 0,Y 212.015,Z 673.707,A -85,B 0,C 180,E1 -20696.199,E2 -20696.199} C_VEL
LIN {X 0,Y 211.778,Z 670.818,A -85,B 0,C 180,E1 -20699.049,E2 -20699.049} C_VEL
LIN {X 0,Y 211.707,Z 667.078,A -85,B 0,C 180,E1 -20701.903,E2 -20701.903} C_VEL
LIN {X 0,Y 211.854,Z 660.657,A -85,B 0,C 180,E1 -20705.712,E2 -20705.712} C_VEL
LIN {X 0,Y 212.313,Z 653.51,A -85,B 0,C 180,E1 -20709.047,E2 -20709.047} C_VEL
LIN {X 0,Y 213.106,Z 644.712,A -85,B 0,C 180,E1 -20712.378,E2 -20712.378} C_VEL
LIN {X 0,Y 214.157,Z 635.598,A -85,B 0,C 180,E1 -20715.221,E2 -20715.221} C_VEL
LIN {X 0,Y 215.252,Z 626.629,A -85,B 0,C 180,E1 -20717.579,E2 -20717.579} C_VEL
LIN {X 0,Y 216.93,Z 614.359,A -85,B 0,C 180,E1 -20720.299,E2 -20720.299} C_VEL
LIN {X 0,Y 218.617,Z 601.126,A -85,B 0,C 180,E1 -20722.692,E2 -20722.692} C_VEL
LIN {X 0,Y 220.568,Z 587.317,A -85,B 0,C 180,E1 -20724.721,E2 -20724.721} C_VEL
LIN {X 0,Y 222.31,Z 572.096,A -85,B 0,C 180,E1 -20726.522,E2 -20726.522} C_VEL
LIN {X 0,Y 223.901,Z 556.189,A -85,B 0,C 180,E1 -20727.961,E2 -20727.961} C_VEL
LIN {X 0,Y 225.23,Z 539.76,A -85,B 0,C 180,E1 -20729.056,E2 -20729.056} C_VEL
LIN {X 0,Y 231.975,Z 447.038,A -85,B 0,C 180,E1 -20733.851,E2 -20733.851} C_VEL
LIN {X 0,Y 230.316,Z 432.417,A -85,B 0,C 180,E1 -20734.899,E2 -20734.899} C_VEL
LIN {X 0,Y 230.236,Z 430.768,A -85,B 0,C 180,E1 -20735.251,E2 -20735.251} C_VEL
LIN {X 0,Y 231.373,Z 429.959,A -85,B 0,C 180,E1 -20735.784,E2 -20735.784} C_VEL
LIN {X 0,Y 232.948,Z 428.441,A -85,B 0,C 180,E1 -20736.238,E2 -20736.238} C_VEL
LIN {X 0,Y 235.047,Z 424.422,A -85,B 0,C 180,E1 -20736.728,E2 -20736.728} C_VEL
LIN {X 0,Y 237.472,Z 422.482,A -85,B 0,C 180,E1 -20737.407,E2 -20737.407} C_VEL
LIN {X 0,Y 239.197,Z 420.169,A -85,B 0,C 180,E1 -20737.832,E2 -20737.832} C_VEL
LIN {X 0,Y 241.177,Z 423.244,A -85,B 0,C 180,E1 -20738.575,E2 -20738.575} C_VEL
LIN {X 0,Y 247.591,Z 434.531,A -85,B 0,C 180,E1 -20740.885,E2 -20740.885} C_VEL
LIN {X 0,Y 254.57,Z 448.719,A -85,B 0,C 180,E1 -20743.237,E2 -20743.237} C_VEL
LIN {X 0,Y 259.378,Z 460.051,A -85,B 0,C 180,E1 -20744.788,E2 -20744.788} C_VEL
LIN {X 0,Y 254.594,Z 544.289,A -85,B 0,C 180,E1 -20746.972,E2 -20746.972} C_VEL
LIN {X 0,Y 253.1,Z 567.002,A -85,B 0,C 180,E1 -20747.605,E2 -20747.605} C_VEL
LIN {X 0,Y 251.181,Z 582.427,A -85,B 0,C 180,E1 -20748.287,E2 -20748.287} C_VEL
LIN {X 0,Y 248.492,Z 597.85,A -85,B 0,C 180,E1 -20749.287,E2 -20749.287} C_VEL
LIN {X 0,Y 245.63,Z 611.205,A -85,B 0,C 180,E1 -20750.459,E2 -20750.459} C_VEL
LIN {X 0,Y 242.102,Z 625.061,A -85,B 0,C 180,E1 -20752.03,E2 -20752.03} C_VEL
LIN {X 0,Y 238.132,Z 637.827,A -85,B 0,C 180,E1 -20753.824,E2 -20753.824} C_VEL
LIN {X 0,Y 233.959,Z 650.032,A -85,B 0,C 180,E1 -20755.98,E2 -20755.98} C_VEL
LIN {X 0,Y 229.456,Z 662.004,A -85,B 0,C 180,E1 -20758.621,E2 -20758.621} C_VEL
LIN {X 0,Y 225.891,Z 671.242,A -85,B 0,C 180,E1 -20761.168,E2 -20761.168} C_VEL
LIN {X 0,Y 221.987,Z 680.32,A -85,B 0,C 180,E1 -20764.194,E2 -20764.194} C_VEL
LIN {X 0,Y 218.829,Z 687.858,A -85,B 0,C 180,E1 -20767.331,E2 -20767.331} C_VEL
LIN {X 0,Y 215.926,Z 694.888,A -85,B 0,C 180,E1 -20771.005,E2 -20771.005} C_VEL
LIN {X 0,Y 213.839,Z 700.417,A -85,B 0,C 180,E1 -20774.756,E2 -20774.756} C_VEL
LIN {X 0,Y 212.394,Z 704.601,A -85,B 0,C 180,E1 -20778.548,E2 -20778.548} C_VEL
LIN {X 0,Y 211.624,Z 707.539,A -85,B 0,C 180,E1 -20782.366,E2 -20782.366} C_VEL
LIN {X 0,Y 211.349,Z 709.299,A -85,B 0,C 180,E1 -20786.186,E2 -20786.186} C_VEL
LIN {X 0,Y 211.391,Z 709.907,A -85,B 0,C 180,E1 -20790,E2 -20790} C_VEL
LIN {X 0,Y 211.337,Z 709.302,A -85,B 0,C 180,E1 -20793.927,E2 -20793.927} C_VEL
LIN {X 0,Y 211.623,Z 707.614,A -85,B 0,C 180,E1 -20797.633,E2 -20797.633} C_VEL
LIN {X 0,Y 212.384,Z 704.725,A -85,B 0,C 180,E1 -20801.452,E2 -20801.452} C_VEL
LIN {X 0,Y 213.807,Z 700.595,A -85,B 0,C 180,E1 -20805.246,E2 -20805.246} C_VEL
LIN {X 0,Y 215.851,Z 695.114,A -85,B 0,C 180,E1 -20809.001,E2 -20809.001} C_VEL
LIN {X 0,Y 218.757,Z 688.133,A -85,B 0,C 180,E1 -20812.676,E2 -20812.676} C_VEL
LIN {X 0,Y 221.889,Z 680.658,A -85,B 0,C 180,E1 -20815.818,E2 -20815.818} C_VEL
LIN {X 0,Y 225.792,Z 671.653,A -85,B 0,C 180,E1 -20818.846,E2 -20818.846} C_VEL
LIN {X 0,Y 229.349,Z 662.452,A -85,B 0,C 180,E1 -20821.395,E2 -20821.395} C_VEL
LIN {X 0,Y 233.879,Z 650.605,A -85,B 0,C 180,E1 -20824.033,E2 -20824.033} C_VEL
LIN {X 0,Y 238.033,Z 638.515,A -85,B 0,C 180,E1 -20826.193,E2 -20826.193} C_VEL
LIN {X 0,Y 242.166,Z 625.152,A -85,B 0,C 180,E1 -20828.087,E2 -20828.087} C_VEL
LIN {X 0,Y 245.515,Z 612.188,A -85,B 0,C 180,E1 -20829.562,E2 -20829.562} C_VEL
LIN {X 0,Y 248.577,Z 597.969,A -85,B 0,C 180,E1 -20830.829,E2 -20830.829} C_VEL
LIN {X 0,Y 251.296,Z 582.599,A -85,B 0,C 180,E1 -20831.823,E2 -20831.823} C_VEL
LIN {X 0,Y 253.2,Z 567.249,A -85,B 0,C 180,E1 -20832.509,E2 -20832.509} C_VEL
LIN {X 0,Y 255.22,Z 535.699,A -85,B 0,C 180,E1 -20833.37,E2 -20833.37} C_VEL
LIN {X 0,Y 259.548,Z 460.213,A -85,B 0,C 180,E1 -20835.317,E2 -20835.317} C_VEL
LIN {X 0,Y 254,Z 447.392,A -85,B 0,C 180,E1 -20837.108,E2 -20837.108} C_VEL
LIN {X 0,Y 247.271,Z 433.779,A -85,B 0,C 180,E1 -20839.396,E2 -20839.396} C_VEL
LIN {X 0,Y 239.696,Z 420.591,A -85,B 0,C 180,E1 -20842.169,E2 -20842.169} C_VEL
LIN {X 0,Y 233.172,Z 410.418,A -85,B 0,C 180,E1 -20844.8,E2 -20844.8} C_VEL
LIN {X 0,Y 228.238,Z 403.357,A -85,B 0,C 180,E1 -20846.981,E2 -20846.981} C_VEL
LIN {X 0,Y 224.914,Z 398.815,A -85,B 0,C 180,E1 -20848.571,E2 -20848.571} C_VEL
LIN {X 0,Y 221.815,Z 394.434,A -85,B 0,C 180,E1 -20850.291,E2 -20850.291} C_VEL
LIN {X 0,Y 218.805,Z 388.229,A -85,B 0,C 180,E1 -20854.073,E2 -20854.073} C_VEL
LIN {X 0,Y 215.995,Z 382.709,A -85,B 0,C 180,E1 -20858.026,E2 -20858.026} C_VEL
LIN {X 0,Y 214.072,Z 379.614,A -85,B 0,C 180,E1 -20860.834,E2 -20860.834} C_VEL
LIN {X 0,Y 213.878,Z 378.502,A -85,B 0,C 180,E1 -20862.029,E2 -20862.029} C_VEL
LIN {X 0,Y 213.937,Z 378.452,A -85,B 0,C 180,E1 -20866.705,E2 -20866.705} C_VEL
LIN {X 0,Y 214.126,Z 378.41,A -85,B 0,C 180,E1 -20870.13,E2 -20870.13} C_VEL
LIN {X 0,Y 213.503,Z 378.51,A -85,B 0,C 180,E1 -20871.698,E2 -20871.698} C_VEL
LIN {X 0,Y 210.747,Z 378.867,A -85,B 0,C 180,E1 -20874.261,E2 -20874.261} C_VEL
LIN {X 0,Y 208.413,Z 379.159,A -85,B 0,C 180,E1 -20876.355,E2 -20876.355} C_VEL
LIN {X 0,Y 207.447,Z 379.266,A -85,B 0,C 180,E1 -20877.979,E2 -20877.979} C_VEL
LIN {X 0,Y 207.387,Z 379.266,A -85,B 0,C 180,E1 -20878.529,E2 -20878.529} C_VEL
LIN {X 0,Y 207.511,Z 379.235,A -85,B 0,C 180,E1 -20880,E2 -20880} C_VEL
LIN {X 0,Y 207.379,Z 379.243,A -85,B 0,C 180,E1 -20881.942,E2 -20881.942} C_VEL
LIN {X 0,Y 207.127,Z 379.273,A -85,B 0,C 180,E1 -20887.8,E2 -20887.8} C_VEL
LIN {X 0,Y 206.916,Z 379.317,A -85,B 0,C 180,E1 -20891.759,E2 -20891.759} C_VEL
LIN {X 0,Y 206.882,Z 379.447,A -85,B 0,C 180,E1 -20894.258,E2 -20894.258} C_VEL
LIN {X 0,Y 207.094,Z 380.502,A -85,B 0,C 180,E1 -20895.753,E2 -20895.753} C_VEL
LIN {X 0,Y 209.982,Z 384.674,A -85,B 0,C 180,E1 -20900.422,E2 -20900.422} C_VEL
LIN {X 0,Y 212.078,Z 388.519,A -85,B 0,C 180,E1 -20903.432,E2 -20903.432} C_VEL
LIN {X 0,Y 212.971,Z 389.6,A -85,B 0,C 180,E1 -20904.362,E2 -20904.362} C_VEL
LIN {X 0,Y 215.146,Z 393.395,A -85,B 0,C 180,E1 -20906.821,E2 -20906.821} C_VEL
LIN {X 0,Y 216.617,Z 395.284,A -85,B 0,C 180,E1 -20907.725,E2 -20907.725} C_VEL
LIN {X 0,Y 220.357,Z 399.78,A -85,B 0,C 180,E1 -20909.824,E2 -20909.824} C_VEL
LIN {X 0,Y 223.103,Z 403.228,A -85,B 0,C 180,E1 -20911.251,E2 -20911.251} C_VEL
LIN {X 0,Y 230.425,Z 413.058,A -85,B 0,C 180,E1 -20914.682,E2 -20914.682} C_VEL
LIN {X 0,Y 237.53,Z 423.444,A -85,B 0,C 180,E1 -20917.607,E2 -20917.607} C_VEL
LIN {X 0,Y 245.649,Z 436.593,A -85,B 0,C 180,E1 -20920.597,E2 -20920.597} C_VEL
LIN {X 0,Y 252.982,Z 455.702,A -85,B 0,C 180,E1 -20923.29,E2 -20923.29} C_VEL
LIN {X 0,Y 254.091,Z 458.764,A -85,B 0,C 180,E1 -20923.679,E2 -20923.679} C_VEL
LIN {X 0,Y 248.021,Z 561.403,A -85,B 0,C 180,E1 -20926.385,E2 -20926.385} C_VEL
LIN {X 0,Y 246.484,Z 576.287,A -85,B 0,C 180,E1 -20926.959,E2 -20926.959} C_VEL
LIN {X 0,Y 244.235,Z 590.303,A -85,B 0,C 180,E1 -20927.73,E2 -20927.73} C_VEL
LIN {X 0,Y 241.392,Z 604.281,A -85,B 0,C 180,E1 -20928.798,E2 -20928.798} C_VEL
LIN {X 0,Y 238.025,Z 618.202,A -85,B 0,C 180,E1 -20930.22,E2 -20930.22} C_VEL
LIN {X 0,Y 234.022,Z 631.911,A -85,B 0,C 180,E1 -20932.002,E2 -20932.002} C_VEL
LIN {X 0,Y 229.893,Z 643.99,A -85,B 0,C 180,E1 -20933.951,E2 -20933.951} C_VEL
LIN {X 0,Y 225.404,Z 656.016,A -85,B 0,C 180,E1 -20936.397,E2 -20936.397} C_VEL
LIN {X 0,Y 221.241,Z 666.116,A -85,B 0,C 180,E1 -20938.922,E2 -20938.922} C_VEL
LIN {X 0,Y 217.204,Z 675.961,A -85,B 0,C 180,E1 -20942.02,E2 -20942.02} C_VEL
LIN {X 0,Y 213.514,Z 684.128,A -85,B 0,C 180,E1 -20945.186,E2 -20945.186} C_VEL
LIN {X 0,Y 210.527,Z 690.879,A -85,B 0,C 180,E1 -20948.456,E2 -20948.456} C_VEL
LIN {X 0,Y 207.873,Z 697.131,A -85,B 0,C 180,E1 -20952.285,E2 -20952.285} C_VEL
LIN {X 0,Y 206.004,Z 701.953,A -85,B 0,C 180,E1 -20956.184,E2 -20956.184} C_VEL
LIN {X 0,Y 204.917,Z 705.476,A -85,B 0,C 180,E1 -20960.126,E2 -20960.126} C_VEL
LIN {X 0,Y 204.388,Z 707.793,A -85,B 0,C 180,E1 -20964.079,E2 -20964.079} C_VEL
LIN {X 0,Y 204.293,Z 708.955,A -85,B 0,C 180,E1 -20968.029,E2 -20968.029} C_VEL
LIN {X 0,Y 204.293,Z 708.952,A -85,B 0,C 180,E1 -20971.972,E2 -20971.972} C_VEL
LIN {X 0,Y 204.389,Z 707.777,A -85,B 0,C 180,E1 -20975.921,E2 -20975.921} C_VEL
LIN {X 0,Y 204.917,Z 705.444,A -85,B 0,C 180,E1 -20979.874,E2 -20979.874} C_VEL
LIN {X 0,Y 206.007,Z 701.898,A -85,B 0,C 180,E1 -20983.816,E2 -20983.816} C_VEL
LIN {X 0,Y 207.871,Z 697.055,A -85,B 0,C 180,E1 -20987.715,E2 -20987.715} C_VEL
LIN {X 0,Y 210.538,Z 690.803,A -85,B 0,C 180,E1 -20991.543,E2 -20991.543} C_VEL
LIN {X 0,Y 211.322,Z 689.273,A -85,B 0,C 180,E1 -20992.486,E2 -20992.486} C_VEL
LIN {X 0,Y 214.328,Z 686.9,A -85,B 0,C 180,E1 -20995.232,E2 -20995.232} C_VEL
LIN {X 0,Y 220.688,Z 681.624,A -85,B 0,C 180,E1 -20999.578,E2 -20999.578} C_VEL
LIN {X 0,Y 226.856,Z 676.251,A -85,B 0,C 180,E1 -21002.83,E2 -21002.83} C_VEL
LIN {X 0,Y 233.977,Z 669.699,A -85,B 0,C 180,E1 -21005.853,E2 -21005.853} C_VEL
LIN {X 0,Y 243.024,Z 660.934,A -85,B 0,C 180,E1 -21008.976,E2 -21008.976} C_VEL
LIN {X 0,Y 251.962,Z 651.68,A -85,B 0,C 180,E1 -21011.488,E2 -21011.488} C_VEL
LIN {X 0,Y 260.439,Z 642.269,A -85,B 0,C 180,E1 -21013.482,E2 -21013.482} C_VEL
LIN {X 0,Y 269.451,Z 631.503,A -85,B 0,C 180,E1 -21015.297,E2 -21015.297} C_VEL
LIN {X 0,Y 277.798,Z 620.665,A -85,B 0,C 180,E1 -21016.718,E2 -21016.718} C_VEL
LIN {X 0,Y 278.009,Z 620.322,A -85,B 0,C 180,E1 -21016.957,E2 -21016.957} C_VEL
LIN {X 0,Y 268.83,Z 631.559,A -85,B 0,C 180,E1 -21018.692,E2 -21018.692} C_VEL
LIN {X 0,Y 260.131,Z 641.197,A -85,B 0,C 180,E1 -21020.587,E2 -21020.587} C_VEL
LIN {X 0,Y 252.023,Z 649.426,A -85,B 0,C 180,E1 -21022.661,E2 -21022.661} C_VEL
LIN {X 0,Y 242.466,Z 658.291,A -85,B 0,C 180,E1 -21025.583,E2 -21025.583} C_VEL
LIN {X 0,Y 234.771,Z 664.706,A -85,B 0,C 180,E1 -21028.408,E2 -21028.408} C_VEL
LIN {X 0,Y 227.799,Z 669.871,A -85,B 0,C 180,E1 -21031.432,E2 -21031.432} C_VEL
LIN {X 0,Y 223.107,Z 672.934,A -85,B 0,C 180,E1 -21033.832,E2 -21033.832} C_VEL
LIN {X 0,Y 217.803,Z 675.962,A -85,B 0,C 180,E1 -21037.219,E2 -21037.219} C_VEL
LIN {X 0,Y 213.368,Z 677.847,A -85,B 0,C 180,E1 -21040.769,E2 -21040.769} C_VEL
LIN {X 0,Y 210.03,Z 678.54,A -85,B 0,C 180,E1 -21044.473,E2 -21044.473} C_VEL
LIN {X 0,Y 207.432,Z 678.064,A -85,B 0,C 180,E1 -21048.271,E2 -21048.271} C_VEL
LIN {X 0,Y 205.743,Z 676.376,A -85,B 0,C 180,E1 -21052.147,E2 -21052.147} C_VEL
LIN {X 0,Y 204.945,Z 673.428,A -85,B 0,C 180,E1 -21056.068,E2 -21056.068} C_VEL
LIN {X 0,Y 204.714,Z 670.329,A -85,B 0,C 180,E1 -21059.017,E2 -21059.017} C_VEL
LIN {X 0,Y 204.646,Z 666.386,A -85,B 0,C 180,E1 -21061.968,E2 -21061.968} C_VEL
LIN {X 0,Y 204.811,Z 659.68,A -85,B 0,C 180,E1 -21065.909,E2 -21065.909} C_VEL
LIN {X 0,Y 205.318,Z 652.211,A -85,B 0,C 180,E1 -21069.358,E2 -21069.358} C_VEL
LIN {X 0,Y 206.158,Z 643.02,A -85,B 0,C 180,E1 -21072.803,E2 -21072.803} C_VEL
LIN {X 0,Y 207.533,Z 631.806,A -85,B 0,C 180,E1 -21076.224,E2 -21076.224} C_VEL
LIN {X 0,Y 209.027,Z 620.158,A -85,B 0,C 180,E1 -21079.137,E2 -21079.137} C_VEL
LIN {X 0,Y 210.757,Z 607.213,A -85,B 0,C 180,E1 -21081.776,E2 -21081.776} C_VEL
LIN {X 0,Y 212.705,Z 593.044,A -85,B 0,C 180,E1 -21084.135,E2 -21084.135} C_VEL
LIN {X 0,Y 214.484,Z 579.259,A -85,B 0,C 180,E1 -21085.993,E2 -21085.993} C_VEL
LIN {X 0,Y 216.134,Z 564.143,A -85,B 0,C 180,E1 -21087.605,E2 -21087.605} C_VEL
LIN {X 0,Y 217.715,Z 547.203,A -85,B 0,C 180,E1 -21088.961,E2 -21088.961} C_VEL
LIN {X 0,Y 224.853,Z 454.261,A -85,B 0,C 180,E1 -21094.101,E2 -21094.101} C_VEL
LIN {X 0,Y 225.844,Z 448.344,A -85,B 0,C 180,E1 -21094.685,E2 -21094.685} C_VEL
LIN {X 0,Y 227.555,Z 446.96,A -85,B 0,C 180,E1 -21095.351,E2 -21095.351} C_VEL
LIN {X 0,Y 229.472,Z 443.676,A -85,B 0,C 180,E1 -21095.846,E2 -21095.846} C_VEL
LIN {X 0,Y 232.003,Z 436.663,A -85,B 0,C 180,E1 -21096.342,E2 -21096.342} C_VEL
LIN {X 0,Y 234.431,Z 434.716,A -85,B 0,C 180,E1 -21097.042,E2 -21097.042} C_VEL
LIN {X 0,Y 236.715,Z 431.413,A -85,B 0,C 180,E1 -21097.605,E2 -21097.605} C_VEL
LIN {X 0,Y 237.723,Z 429.783,A -85,B 0,C 180,E1 -21097.84,E2 -21097.84} C_VEL
LIN {X 0,Y 238.295,Z 429.47,A -85,B 0,C 180,E1 -21098,E2 -21098} C_VEL
LIN {X 0,Y 244.098,Z 440.054,A -85,B 0,C 180,E1 -21100.18,E2 -21100.18} C_VEL
LIN {X 0,Y 250.302,Z 452.92,A -85,B 0,C 180,E1 -21102.367,E2 -21102.367} C_VEL
LIN {X 0,Y 254.269,Z 462.262,A -85,B 0,C 180,E1 -21103.71,E2 -21103.71} C_VEL
LIN {X 0,Y 249.799,Z 538.828,A -85,B 0,C 180,E1 -21105.726,E2 -21105.726} C_VEL
LIN {X 0,Y 247.906,Z 566.931,A -85,B 0,C 180,E1 -21106.499,E2 -21106.499} C_VEL
LIN {X 0,Y 245.94,Z 582.382,A -85,B 0,C 180,E1 -21107.189,E2 -21107.189} C_VEL
LIN {X 0,Y 243.155,Z 597.817,A -85,B 0,C 180,E1 -21108.196,E2 -21108.196} C_VEL
LIN {X 0,Y 240.184,Z 611.177,A -85,B 0,C 180,E1 -21109.378,E2 -21109.378} C_VEL
LIN {X 0,Y 236.486,Z 625.224,A -85,B 0,C 180,E1 -21110.995,E2 -21110.995} C_VEL
LIN {X 0,Y 232.01,Z 639.003,A -85,B 0,C 180,E1 -21112.983,E2 -21112.983} C_VEL
LIN {X 0,Y 227.696,Z 651.014,A -85,B 0,C 180,E1 -21115.179,E2 -21115.179} C_VEL
LIN {X 0,Y 223.388,Z 661.987,A -85,B 0,C 180,E1 -21117.667,E2 -21117.667} C_VEL
LIN {X 0,Y 219.635,Z 671.226,A -85,B 0,C 180,E1 -21120.265,E2 -21120.265} C_VEL
LIN {X 0,Y 215.571,Z 680.306,A -85,B 0,C 180,E1 -21123.367,E2 -21123.367} C_VEL
LIN {X 0,Y 212.228,Z 687.844,A -85,B 0,C 180,E1 -21126.585,E2 -21126.585} C_VEL
LIN {X 0,Y 209.152,Z 694.874,A -85,B 0,C 180,E1 -21130.365,E2 -21130.365} C_VEL
LIN {X 0,Y 206.944,Z 700.404,A -85,B 0,C 180,E1 -21134.235,E2 -21134.235} C_VEL
LIN {X 0,Y 205.397,Z 704.587,A -85,B 0,C 180,E1 -21138.153,E2 -21138.153} C_VEL
LIN {X 0,Y 204.562,Z 707.526,A -85,B 0,C 180,E1 -21142.101,E2 -21142.101} C_VEL
LIN {X 0,Y 204.257,Z 709.325,A -85,B 0,C 180,E1 -21146.22,E2 -21146.22} C_VEL
LIN {X 0,Y 204.297,Z 709.893,A -85,B 0,C 180,E1 -21150,E2 -21150} C_VEL
LIN {X 0,Y 204.258,Z 709.316,A -85,B 0,C 180,E1 -21153.946,E2 -21153.946} C_VEL
LIN {X 0,Y 204.562,Z 707.599,A -85,B 0,C 180,E1 -21157.899,E2 -21157.899} C_VEL
LIN {X 0,Y 205.387,Z 704.71,A -85,B 0,C 180,E1 -21161.847,E2 -21161.847} C_VEL
LIN {X 0,Y 206.911,Z 700.58,A -85,B 0,C 180,E1 -21165.767,E2 -21165.767} C_VEL
LIN {X 0,Y 209.164,Z 694.819,A -85,B 0,C 180,E1 -21169.811,E2 -21169.811} C_VEL
LIN {X 0,Y 212.155,Z 688.115,A -85,B 0,C 180,E1 -21173.423,E2 -21173.423} C_VEL
LIN {X 0,Y 215.483,Z 680.639,A -85,B 0,C 180,E1 -21176.645,E2 -21176.645} C_VEL
LIN {X 0,Y 219.509,Z 671.713,A -85,B 0,C 180,E1 -21179.724,E2 -21179.724} C_VEL
LIN {X 0,Y 223.284,Z 662.43,A -85,B 0,C 180,E1 -21182.35,E2 -21182.35} C_VEL
LIN {X 0,Y 228.018,Z 650.58,A -85,B 0,C 180,E1 -21185.034,E2 -21185.034} C_VEL
LIN {X 0,Y 232.319,Z 638.487,A -85,B 0,C 180,E1 -21187.231,E2 -21187.231} C_VEL
LIN {X 0,Y 236.266,Z 626.263,A -85,B 0,C 180,E1 -21188.997,E2 -21188.997} C_VEL
LIN {X 0,Y 239.621,Z 613.876,A -85,B 0,C 180,E1 -21190.46,E2 -21190.46} C_VEL
LIN {X 0,Y 242.77,Z 600.112,A -85,B 0,C 180,E1 -21191.746,E2 -21191.746} C_VEL
LIN {X 0,Y 245.548,Z 585.475,A -85,B 0,C 180,E1 -21192.755,E2 -21192.755} C_VEL
LIN {X 0,Y 247.659,Z 570.408,A -85,B 0,C 180,E1 -21193.484,E2 -21193.484} C_VEL
LIN {X 0,Y 249.013,Z 553.412,A -85,B 0,C 180,E1 -21194.027,E2 -21194.027} C_VEL
LIN {X 0,Y 254.446,Z 462.501,A -85,B 0,C 180,E1 -21196.392,E2 -21196.392} C_VEL
LIN {X 0,Y 249.246,Z 450.481,A -85,B 0,C 180,E1 -21198.161,E2 -21198.161} C_VEL
LIN {X 0,Y 242.04,Z 435.92,A -85,B 0,C 180,E1 -21200.756,E2 -21200.756} C_VEL
LIN {X 0,Y 234.246,Z 422.393,A -85,B 0,C 180,E1 -21203.819,E2 -21203.819} C_VEL
LIN {X 0,Y 227.533,Z 412.023,A -85,B 0,C 180,E1 -21206.763,E2 -21206.763} C_VEL
LIN {X 0,Y 222.545,Z 405.071,A -85,B 0,C 180,E1 -21209.19,E2 -21209.19} C_VEL
LIN {X 0,Y 218.428,Z 399.584,A -85,B 0,C 180,E1 -21211.405,E2 -21211.405} C_VEL
LIN {X 0,Y 214.57,Z 394.363,A -85,B 0,C 180,E1 -21213.835,E2 -21213.835} C_VEL
LIN {X 0,Y 211.266,Z 387.855,A -85,B 0,C 180,E1 -21218.662,E2 -21218.662} C_VEL
LIN {X 0,Y 209.121,Z 383.728,A -85,B 0,C 180,E1 -21222.394,E2 -21222.394} C_VEL
LIN {X 0,Y 207.118,Z 380.516,A -85,B 0,C 180,E1 -21226.259,E2 -21226.259} C_VEL
LIN {X 0,Y 206.917,Z 379.46,A -85,B 0,C 180,E1 -21227.744,E2 -21227.744} C_VEL
LIN {X 0,Y 207.1,Z 379.285,A -85,B 0,C 180,E1 -21230.231,E2 -21230.231} C_VEL
LIN {X 0,Y 207.052,Z 379.288,A -85,B 0,C 180,E1 -21234.155,E2 -21234.155} C_VEL
LIN {X 0,Y 207.387,Z 379.266,A -85,B 0,C 180,E1 -21238.529,E2 -21238.529} C_VEL
LIN {X 0,Y 206.733,Z 379.415,A -85,B 0,C 180,E1 -21240.147,E2 -21240.147} C_VEL
LIN {X 0,Y 205.111,Z 379.847,A -85,B 0,C 180,E1 -21241.734,E2 -21241.734} C_VEL
LIN {X 0,Y 201.393,Z 381.153,A -85,B 0,C 180,E1 -21244.935,E2 -21244.935} C_VEL
LIN {X 0,Y 200.511,Z 381.836,A -85,B 0,C 180,E1 -21246.61,E2 -21246.61} C_VEL
LIN {X 0,Y 200.522,Z 382.043,A -85,B 0,C 180,E1 -21247.176,E2 -21247.176} C_VEL
LIN {X 0,Y 202.839,Z 385.234,A -85,B 0,C 180,E1 -21254.036,E2 -21254.036} C_VEL
LIN {X 0,Y 206.047,Z 390.423,A -85,B 0,C 180,E1 -21259.943,E2 -21259.943} C_VEL
LIN {X 0,Y 207.809,Z 393.761,A -85,B 0,C 180,E1 -21262.494,E2 -21262.494} C_VEL
LIN {X 0,Y 210.549,Z 396.844,A -85,B 0,C 180,E1 -21264.499,E2 -21264.499} C_VEL
LIN {X 0,Y 214.187,Z 401.159,A -85,B 0,C 180,E1 -21266.884,E2 -21266.884} C_VEL
LIN {X 0,Y 218.072,Z 406.064,A -85,B 0,C 180,E1 -21269.173,E2 -21269.173} C_VEL
LIN {X 0,Y 222.655,Z 412.077,A -85,B 0,C 180,E1 -21271.598,E2 -21271.598} C_VEL
LIN {X 0,Y 228.14,Z 419.751,A -85,B 0,C 180,E1 -21274.208,E2 -21274.208} C_VEL
LIN {X 0,Y 234.258,Z 428.874,A -85,B 0,C 180,E1 -21276.823,E2 -21276.823} C_VEL
LIN {X 0,Y 241.829,Z 441.419,A -85,B 0,C 180,E1 -21279.744,E2 -21279.744} C_VEL
LIN {X 0,Y 248.634,Z 459.625,A -85,B 0,C 180,E1 -21282.375,E2 -21282.375} C_VEL
LIN {X 0,Y 249.101,Z 460.997,A -85,B 0,C 180,E1 -21282.55,E2 -21282.55} C_VEL
LIN {X 0,Y 242.794,Z 562.96,A -85,B 0,C 180,E1 -21285.271,E2 -21285.271} C_VEL
LIN {X 0,Y 241.071,Z 578.144,A -85,B 0,C 180,E1 -21285.891,E2 -21285.891} C_VEL
LIN {X 0,Y 238.527,Z 592.906,A -85,B 0,C 180,E1 -21286.761,E2 -21286.761} C_VEL
LIN {X 0,Y 235.626,Z 606.279,A -85,B 0,C 180,E1 -21287.848,E2 -21287.848} C_VEL
LIN {X 0,Y 232.413,Z 618.886,A -85,B 0,C 180,E1 -21289.177,E2 -21289.177} C_VEL
LIN {X 0,Y 228.447,Z 631.941,A -85,B 0,C 180,E1 -21290.901,E2 -21290.901} C_VEL
LIN {X 0,Y 224.186,Z 644.016,A -85,B 0,C 180,E1 -21292.882,E2 -21292.882} C_VEL
LIN {X 0,Y 219.5,Z 656.039,A -85,B 0,C 180,E1 -21295.367,E2 -21295.367} C_VEL
LIN {X 0,Y 215.17,Z 666.137,A -85,B 0,C 180,E1 -21297.943,E2 -21297.943} C_VEL
LIN {X 0,Y 210.928,Z 675.98,A -85,B 0,C 180,E1 -21301.11,E2 -21301.11} C_VEL
LIN {X 0,Y 207.031,Z 684.146,A -85,B 0,C 180,E1 -21304.354,E2 -21304.354} C_VEL
LIN {X 0,Y 203.869,Z 690.896,A -85,B 0,C 180,E1 -21307.716,E2 -21307.716} C_VEL
LIN {X 0,Y 201.069,Z 697.147,A -85,B 0,C 180,E1 -21311.665,E2 -21311.665} C_VEL
LIN {X 0,Y 199.067,Z 701.968,A -85,B 0,C 180,E1 -21315.692,E2 -21315.692} C_VEL
LIN {X 0,Y 197.894,Z 705.491,A -85,B 0,C 180,E1 -21319.772,E2 -21319.772} C_VEL
LIN {X 0,Y 197.303,Z 707.807,A -85,B 0,C 180,E1 -21323.866,E2 -21323.866} C_VEL
LIN {X 0,Y 197.204,Z 708.969,A -85,B 0,C 180,E1 -21327.958,E2 -21327.958} C_VEL
LIN {X 0,Y 197.204,Z 708.965,A -85,B 0,C 180,E1 -21332.043,E2 -21332.043} C_VEL
LIN {X 0,Y 197.304,Z 707.79,A -85,B 0,C 180,E1 -21336.135,E2 -21336.135} C_VEL
LIN {X 0,Y 197.895,Z 705.458,A -85,B 0,C 180,E1 -21340.228,E2 -21340.228} C_VEL
LIN {X 0,Y 199.07,Z 701.911,A -85,B 0,C 180,E1 -21344.308,E2 -21344.308} C_VEL
LIN {X 0,Y 201.067,Z 697.069,A -85,B 0,C 180,E1 -21348.336,E2 -21348.336} C_VEL
LIN {X 0,Y 203.882,Z 690.823,A -85,B 0,C 180,E1 -21352.283,E2 -21352.283} C_VEL
LIN {X 0,Y 204.503,Z 689.633,A -85,B 0,C 180,E1 -21353.012,E2 -21353.012} C_VEL
LIN {X 0,Y 210.404,Z 685.572,A -85,B 0,C 180,E1 -21357.881,E2 -21357.881} C_VEL
LIN {X 0,Y 216.069,Z 681.399,A -85,B 0,C 180,E1 -21361.361,E2 -21361.361} C_VEL
LIN {X 0,Y 222.743,Z 676.138,A -85,B 0,C 180,E1 -21364.607,E2 -21364.607} C_VEL
LIN {X 0,Y 230.442,Z 669.777,A -85,B 0,C 180,E1 -21367.587,E2 -21367.587} C_VEL
LIN {X 0,Y 240.032,Z 661.265,A -85,B 0,C 180,E1 -21370.653,E2 -21370.653} C_VEL
LIN {X 0,Y 249.46,Z 652.307,A -85,B 0,C 180,E1 -21373.094,E2 -21373.094} C_VEL
LIN {X 0,Y 258.31,Z 643.253,A -85,B 0,C 180,E1 -21375.024,E2 -21375.024} C_VEL
LIN {X 0,Y 266.615,Z 634.156,A -85,B 0,C 180,E1 -21376.571,E2 -21376.571} C_VEL
LIN {X 0,Y 268.158,Z 632.293,A -85,B 0,C 180,E1 -21377.046,E2 -21377.046} C_VEL
LIN {X 0,Y 257.766,Z 643.021,A -85,B 0,C 180,E1 -21379.129,E2 -21379.129} C_VEL
LIN {X 0,Y 248.086,Z 652.028,A -85,B 0,C 180,E1 -21381.447,E2 -21381.447} C_VEL
LIN {X 0,Y 239.161,Z 659.531,A -85,B 0,C 180,E1 -21384.005,E2 -21384.005} C_VEL
LIN {X 0,Y 230.993,Z 665.724,A -85,B 0,C 180,E1 -21386.794,E2 -21386.794} C_VEL
LIN {X 0,Y 223.581,Z 670.721,A -85,B 0,C 180,E1 -21389.805,E2 -21389.805} C_VEL
LIN {X 0,Y 216.931,Z 674.531,A -85,B 0,C 180,E1 -21393.028,E2 -21393.028} C_VEL
LIN {X 0,Y 211.393,Z 677.151,A -85,B 0,C 180,E1 -21396.487,E2 -21396.487} C_VEL
LIN {X 0,Y 206.729,Z 678.665,A -85,B 0,C 180,E1 -21400.126,E2 -21400.126} C_VEL
LIN {X 0,Y 203.226,Z 679.036,A -85,B 0,C 180,E1 -21403.939,E2 -21403.939} C_VEL
LIN {X 0,Y 200.504,Z 678.268,A -85,B 0,C 180,E1 -21407.86,E2 -21407.86} C_VEL
LIN {X 0,Y 198.58,Z 676.007,A -85,B 0,C 180,E1 -21412.29,E2 -21412.29} C_VEL
LIN {X 0,Y 197.878,Z 673.073,A -85,B 0,C 180,E1 -21415.927,E2 -21415.927} C_VEL
LIN {X 0,Y 197.652,Z 669.741,A -85,B 0,C 180,E1 -21418.982,E2 -21418.982} C_VEL
LIN {X 0,Y 197.587,Z 665.574,A -85,B 0,C 180,E1 -21422.039,E2 -21422.039} C_VEL
LIN {X 0,Y 197.726,Z 659.545,A -85,B 0,C 180,E1 -21425.592,E2 -21425.592} C_VEL
LIN {X 0,Y 198.225,Z 651.96,A -85,B 0,C 180,E1 -21429.181,E2 -21429.181} C_VEL
LIN {X 0,Y 199.056,Z 642.665,A -85,B 0,C 180,E1 -21432.748,E2 -21432.748} C_VEL
LIN {X 0,Y 200.222,Z 633.1,A -85,B 0,C 180,E1 -21435.786,E2 -21435.786} C_VEL
LIN {X 0,Y 201.703,Z 621.665,A -85,B 0,C 180,E1 -21438.802,E2 -21438.802} C_VEL
LIN {X 0,Y 203.377,Z 609.466,A -85,B 0,C 180,E1 -21441.461,E2 -21441.461} C_VEL
LIN {X 0,Y 205.314,Z 595.245,A -85,B 0,C 180,E1 -21443.985,E2 -21443.985} C_VEL
LIN {X 0,Y 207.119,Z 581.925,A -85,B 0,C 180,E1 -21445.905,E2 -21445.905} C_VEL
LIN {X 0,Y 208.893,Z 566.416,A -85,B 0,C 180,E1 -21447.692,E2 -21447.692} C_VEL
LIN {X 0,Y 210.41,Z 550.165,A -85,B 0,C 180,E1 -21449.105,E2 -21449.105} C_VEL
LIN {X 0,Y 212.193,Z 527.679,A -85,B 0,C 180,E1 -21450.502,E2 -21450.502} C_VEL
LIN {X 0,Y 214.843,Z 494.581,A -85,B 0,C 180,E1 -21452.459,E2 -21452.459} C_VEL
LIN {X 0,Y 215.648,Z 489.105,A -85,B 0,C 180,E1 -21453.016,E2 -21453.016} C_VEL
LIN {X 0,Y 216.396,Z 487.211,A -85,B 0,C 180,E1 -21453.373,E2 -21453.373} C_VEL
LIN {X 0,Y 217.74,Z 485.277,A -85,B 0,C 180,E1 -21453.833,E2 -21453.833} C_VEL
LIN {X 0,Y 220.337,Z 479.199,A -85,B 0,C 180,E1 -21454.483,E2 -21454.483} C_VEL
LIN {X 0,Y 223.868,Z 468.04,A -85,B 0,C 180,E1 -21455.169,E2 -21455.169} C_VEL
LIN {X 0,Y 227.79,Z 454.432,A -85,B 0,C 180,E1 -21455.829,E2 -21455.829} C_VEL
LIN {X 0,Y 228.572,Z 453.485,A -85,B 0,C 180,E1 -21456.05,E2 -21456.05} C_VEL
LIN {X 0,Y 230.909,Z 450.709,A -85,B 0,C 180,E1 -21456.695,E2 -21456.695} C_VEL
LIN {X 0,Y 233.502,Z 445.551,A -85,B 0,C 180,E1 -21457.281,E2 -21457.281} C_VEL
LIN {X 0,Y 234.992,Z 441.795,A -85,B 0,C 180,E1 -21457.571,E2 -21457.571} C_VEL
LIN {X 0,Y 236.722,Z 440.105,A -85,B 0,C 180,E1 -21458.028,E2 -21458.028} C_VEL
LIN {X 0,Y 237.941,Z 440.173,A -85,B 0,C 180,E1 -21458.404,E2 -21458.404} C_VEL
LIN {X 0,Y 244.44,Z 453.501,A -85,B 0,C 180,E1 -21460.869,E2 -21460.869} C_VEL
LIN {X 0,Y 249.294,Z 464.763,A -85,B 0,C 180,E1 -21462.609,E2 -21462.609} C_VEL
LIN {X 0,Y 243.852,Z 553.014,A -85,B 0,C 180,E1 -21464.934,E2 -21464.934} C_VEL
LIN {X 0,Y 242.446,Z 570.153,A -85,B 0,C 180,E1 -21465.481,E2 -21465.481} C_VEL
LIN {X 0,Y 240.292,Z 585.287,A -85,B 0,C 180,E1 -21466.22,E2 -21466.22} C_VEL
LIN {X 0,Y 237.421,Z 599.977,A -85,B 0,C 180,E1 -21467.236,E2 -21467.236} C_VEL
LIN {X 0,Y 233.875,Z 614.64,A -85,B 0,C 180,E1 -21468.615,E2 -21468.615} C_VEL
LIN {X 0,Y 229.898,Z 628.608,A -85,B 0,C 180,E1 -21470.346,E2 -21470.346} C_VEL
LIN {X 0,Y 225.536,Z 641.291,A -85,B 0,C 180,E1 -21472.299,E2 -21472.299} C_VEL
LIN {X 0,Y 221.126,Z 652.92,A -85,B 0,C 180,E1 -21474.547,E2 -21474.547} C_VEL
LIN {X 0,Y 216.619,Z 663.739,A -85,B 0,C 180,E1 -21477.137,E2 -21477.137} C_VEL
LIN {X 0,Y 212.812,Z 672.691,A -85,B 0,C 180,E1 -21479.79,E2 -21479.79} C_VEL
LIN {X 0,Y 208.648,Z 681.474,A -85,B 0,C 180,E1 -21482.952,E2 -21482.952} C_VEL
LIN {X 0,Y 204.784,Z 689.754,A -85,B 0,C 180,E1 -21486.754,E2 -21486.754} C_VEL
LIN {X 0,Y 201.783,Z 696.391,A -85,B 0,C 180,E1 -21490.678,E2 -21490.678} C_VEL
LIN {X 0,Y 199.579,Z 701.586,A -85,B 0,C 180,E1 -21494.686,E2 -21494.686} C_VEL
LIN {X 0,Y 198.419,Z 704.574,A -85,B 0,C 180,E1 -21497.73,E2 -21497.73} C_VEL
LIN {X 0,Y 197.501,Z 707.512,A -85,B 0,C 180,E1 -21501.817,E2 -21501.817} C_VEL
LIN {X 0,Y 197.173,Z 709.272,A -85,B 0,C 180,E1 -21505.912,E2 -21505.912} C_VEL
LIN {X 0,Y 197.205,Z 709.88,A -85,B 0,C 180,E1 -21510,E2 -21510} C_VEL
LIN {X 0,Y 197.173,Z 709.302,A -85,B 0,C 180,E1 -21514.088,E2 -21514.088} C_VEL
LIN {X 0,Y 197.5,Z 707.585,A -85,B 0,C 180,E1 -21518.183,E2 -21518.183} C_VEL
LIN {X 0,Y 198.409,Z 704.695,A -85,B 0,C 180,E1 -21522.27,E2 -21522.27} C_VEL
LIN {X 0,Y 200.04,Z 700.564,A -85,B 0,C 180,E1 -21526.323,E2 -21526.323} C_VEL
LIN {X 0,Y 202.316,Z 695.081,A -85,B 0,C 180,E1 -21530.327,E2 -21530.327} C_VEL
LIN {X 0,Y 205.615,Z 688.098,A -85,B 0,C 180,E1 -21534.215,E2 -21534.215} C_VEL
LIN {X 0,Y 209.111,Z 680.621,A -85,B 0,C 180,E1 -21537.524,E2 -21537.524} C_VEL
LIN {X 0,Y 213.182,Z 672,A -85,B 0,C 180,E1 -21540.581,E2 -21540.581} C_VEL
LIN {X 0,Y 217.273,Z 662.408,A -85,B 0,C 180,E1 -21543.359,E2 -21543.359} C_VEL
LIN {X 0,Y 222.212,Z 650.555,A -85,B 0,C 180,E1 -21546.09,E2 -21546.09} C_VEL
LIN {X 0,Y 226.689,Z 638.459,A -85,B 0,C 180,E1 -21548.32,E2 -21548.32} C_VEL
LIN {X 0,Y 231.182,Z 624.852,A -85,B 0,C 180,E1 -21550.297,E2 -21550.297} C_VEL
LIN {X 0,Y 235.189,Z 610.249,A -85,B 0,C 180,E1 -21551.96,E2 -21551.96} C_VEL
LIN {X 0,Y 238.262,Z 596.718,A -85,B 0,C 180,E1 -21553.154,E2 -21553.154} C_VEL
LIN {X 0,Y 241.048,Z 581.632,A -85,B 0,C 180,E1 -21554.115,E2 -21554.115} C_VEL
LIN {X 0,Y 242.949,Z 567.046,A -85,B 0,C 180,E1 -21554.766,E2 -21554.766} C_VEL
LIN {X 0,Y 245.111,Z 535.401,A -85,B 0,C 180,E1 -21555.645,E2 -21555.645} C_VEL
LIN {X 0,Y 249.411,Z 464.89,A -85,B 0,C 180,E1 -21557.514,E2 -21557.514} C_VEL
LIN {X 0,Y 244.304,Z 452.917,A -85,B 0,C 180,E1 -21559.358,E2 -21559.358} C_VEL
LIN {X 0,Y 238.014,Z 440.23,A -85,B 0,C 180,E1 -21561.745,E2 -21561.745} C_VEL
LIN {X 0,Y 230.935,Z 427.645,A -85,B 0,C 180,E1 -21564.674,E2 -21564.674} C_VEL
LIN {X 0,Y 224.641,Z 417.712,A -85,B 0,C 180,E1 -21567.566,E2 -21567.566} C_VEL
LIN {X 0,Y 220.058,Z 411.139,A -85,B 0,C 180,E1 -21569.899,E2 -21569.899} C_VEL
LIN {X 0,Y 216.276,Z 405.937,A -85,B 0,C 180,E1 -21572.02,E2 -21572.02} C_VEL
LIN {X 0,Y 211.294,Z 399.425,A -85,B 0,C 180,E1 -21575.17,E2 -21575.17} C_VEL
LIN {X 0,Y 207.442,Z 394.321,A -85,B 0,C 180,E1 -21578.119,E2 -21578.119} C_VEL
LIN {X 0,Y 205.2,Z 389.976,A -85,B 0,C 180,E1 -21582.046,E2 -21582.046} C_VEL
LIN {X 0,Y 202.635,Z 385.04,A -85,B 0,C 180,E1 -21587.989,E2 -21587.989} C_VEL
LIN {X 0,Y 200.642,Z 382.347,A -85,B 0,C 180,E1 -21593.968,E2 -21593.968} C_VEL
LIN {X 0,Y 200.418,Z 380.695,A -85,B 0,C 180,E1 -21598.562,E2 -21598.562} C_VEL
LIN {X 0,Y 200.518,Z 380.455,A -85,B 0,C 180,E1 -21600,E2 -21600} C_VEL
LIN {X 0,Y 200.228,Z 380.872,A -85,B 0,C 180,E1 -21603.27,E2 -21603.27} C_VEL
LIN {X 0,Y 200.522,Z 382.043,A -85,B 0,C 180,E1 -21607.176,E2 -21607.176} C_VEL
LIN {X 0,Y 200.569,Z 383.235,A -85,B 0,C 180,E1 -21608.826,E2 -21608.826} C_VEL
LIN {X 0,Y 199.969,Z 386.916,A -85,B 0,C 180,E1 -21611.449,E2 -21611.449} C_VEL
LIN {X 0,Y 199.56,Z 391.74,A -85,B 0,C 180,E1 -21614.603,E2 -21614.603} C_VEL
LIN {X 0,Y 199.881,Z 392.9,A -85,B 0,C 180,E1 -21615.695,E2 -21615.695} C_VEL
LIN {X 0,Y 203.885,Z 397.587,A -85,B 0,C 180,E1 -21620.032,E2 -21620.032} C_VEL
LIN {X 0,Y 208.622,Z 403.251,A -85,B 0,C 180,E1 -21623.844,E2 -21623.844} C_VEL
LIN {X 0,Y 212.12,Z 407.537,A -85,B 0,C 180,E1 -21626.238,E2 -21626.238} C_VEL
LIN {X 0,Y 215.766,Z 412.259,A -85,B 0,C 180,E1 -21628.477,E2 -21628.477} C_VEL
LIN {X 0,Y 219.983,Z 417.91,A -85,B 0,C 180,E1 -21630.808,E2 -21630.808} C_VEL
LIN {X 0,Y 225.12,Z 425.263,A -85,B 0,C 180,E1 -21633.369,E2 -21633.369} C_VEL
LIN {X 0,Y 231.416,Z 434.889,A -85,B 0,C 180,E1 -21636.179,E2 -21636.179} C_VEL
LIN {X 0,Y 237.938,Z 445.915,A -85,B 0,C 180,E1 -21638.81,E2 -21638.81} C_VEL
LIN {X 0,Y 244.222,Z 463.13,A -85,B 0,C 180,E1 -21641.374,E2 -21641.374} C_VEL
LIN {X 0,Y 237.821,Z 563.074,A -85,B 0,C 180,E1 -21644.072,E2 -21644.072} C_VEL
LIN {X 0,Y 236.038,Z 578.215,A -85,B 0,C 180,E1 -21644.694,E2 -21644.694} C_VEL
LIN {X 0,Y 233.42,Z 592.958,A -85,B 0,C 180,E1 -21645.571,E2 -21645.571} C_VEL
LIN {X 0,Y 230.402,Z 606.321,A -85,B 0,C 180,E1 -21646.661,E2 -21646.661} C_VEL
LIN {X 0,Y 226.852,Z 619.689,A -85,B 0,C 180,E1 -21648.099,E2 -21648.099} C_VEL
LIN {X 0,Y 222.518,Z 633.249,A -85,B 0,C 180,E1 -21649.945,E2 -21649.945} C_VEL
LIN {X 0,Y 217.676,Z 646.16,A -85,B 0,C 180,E1 -21652.161,E2 -21652.161} C_VEL
LIN {X 0,Y 212.874,Z 657.83,A -85,B 0,C 180,E1 -21654.707,E2 -21654.707} C_VEL
LIN {X 0,Y 207.846,Z 668.822,A -85,B 0,C 180,E1 -21657.708,E2 -21657.708} C_VEL
LIN {X 0,Y 204.081,Z 677.225,A -85,B 0,C 180,E1 -21660.612,E2 -21660.612} C_VEL
LIN {X 0,Y 200.089,Z 685.198,A -85,B 0,C 180,E1 -21663.957,E2 -21663.957} C_VEL
LIN {X 0,Y 196.431,Z 692.623,A -85,B 0,C 180,E1 -21667.934,E2 -21667.934} C_VEL
LIN {X 0,Y 193.686,Z 698.51,A -85,B 0,C 180,E1 -21672.036,E2 -21672.036} C_VEL
LIN {X 0,Y 192.151,Z 701.984,A -85,B 0,C 180,E1 -21675.166,E2 -21675.166} C_VEL
LIN {X 0,Y 190.86,Z 705.506,A -85,B 0,C 180,E1 -21679.391,E2 -21679.391} C_VEL
LIN {X 0,Y 190.221,Z 707.821,A -85,B 0,C 180,E1 -21683.637,E2 -21683.637} C_VEL
LIN {X 0,Y 190.102,Z 708.982,A -85,B 0,C 180,E1 -21687.882,E2 -21687.882} C_VEL
LIN {X 0,Y 190.119,Z 709.133,A -85,B 0,C 180,E1 -21690,E2 -21690} C_VEL
LIN {X 0,Y 190.16,Z 708.534,A -85,B 0,C 180,E1 -21694.239,E2 -21694.239} C_VEL
LIN {X 0,Y 190.459,Z 706.785,A -85,B 0,C 180,E1 -21698.488,E2 -21698.488} C_VEL
LIN {X 0,Y 191.424,Z 703.854,A -85,B 0,C 180,E1 -21702.726,E2 -21702.726} C_VEL
LIN {X 0,Y 193.168,Z 699.672,A -85,B 0,C 180,E1 -21706.922,E2 -21706.922} C_VEL
LIN {X 0,Y 195.632,Z 694.139,A -85,B 0,C 180,E1 -21711.054,E2 -21711.054} C_VEL
LIN {X 0,Y 197.957,Z 689.744,A -85,B 0,C 180,E1 -21713.819,E2 -21713.819} C_VEL
LIN {X 0,Y 201.565,Z 687.716,A -85,B 0,C 180,E1 -21716.954,E2 -21716.954} C_VEL
LIN {X 0,Y 208.549,Z 683.368,A -85,B 0,C 180,E1 -21721.49,E2 -21721.49} C_VEL
LIN {X 0,Y 215.268,Z 678.779,A -85,B 0,C 180,E1 -21724.844,E2 -21724.844} C_VEL
LIN {X 0,Y 223.595,Z 672.7,A -85,B 0,C 180,E1 -21728.147,E2 -21728.147} C_VEL
LIN {X 0,Y 233.795,Z 664.67,A -85,B 0,C 180,E1 -21731.402,E2 -21731.402} C_VEL
LIN {X 0,Y 244.643,Z 655.421,A -85,B 0,C 180,E1 -21734.159,E2 -21734.159} C_VEL
LIN {X 0,Y 253.733,Z 647.007,A -85,B 0,C 180,E1 -21736.068,E2 -21736.068} C_VEL
LIN {X 0,Y 256.442,Z 644.425,A -85,B 0,C 180,E1 -21736.575,E2 -21736.575} C_VEL
LIN {X 0,Y 258.26,Z 642.539,A -85,B 0,C 180,E1 -21737.131,E2 -21737.131} C_VEL
LIN {X 0,Y 247.927,Z 651.601,A -85,B 0,C 180,E1 -21739.309,E2 -21739.309} C_VEL
LIN {X 0,Y 238.373,Z 659.156,A -85,B 0,C 180,E1 -21741.746,E2 -21741.746} C_VEL
LIN {X 0,Y 229.526,Z 665.434,A -85,B 0,C 180,E1 -21744.425,E2 -21744.425} C_VEL
LIN {X 0,Y 221.441,Z 670.516,A -85,B 0,C 180,E1 -21747.348,E2 -21747.348} C_VEL
LIN {X 0,Y 214.063,Z 674.495,A -85,B 0,C 180,E1 -21750.497,E2 -21750.497} C_VEL
LIN {X 0,Y 207.778,Z 677.294,A -85,B 0,C 180,E1 -21753.914,E2 -21753.914} C_VEL
LIN {X 0,Y 202.39,Z 679.02,A -85,B 0,C 180,E1 -21757.544,E2 -21757.544} C_VEL
LIN {X 0,Y 198.161,Z 679.626,A -85,B 0,C 180,E1 -21761.386,E2 -21761.386} C_VEL
LIN {X 0,Y 194.861,Z 679.088,A -85,B 0,C 180,E1 -21765.377,E2 -21765.377} C_VEL
LIN {X 0,Y 192.534,Z 677.401,A -85,B 0,C 180,E1 -21769.484,E2 -21769.484} C_VEL
LIN {X 0,Y 191.12,Z 674.508,A -85,B 0,C 180,E1 -21773.667,E2 -21773.667} C_VEL
LIN {X 0,Y 190.68,Z 670.325,A -85,B 0,C 180,E1 -21777.888,E2 -21777.888} C_VEL
LIN {X 0,Y 190.53,Z 664.656,A -85,B 0,C 180,E1 -21782.114,E2 -21782.114} C_VEL
LIN {X 0,Y 190.674,Z 658.653,A -85,B 0,C 180,E1 -21785.622,E2 -21785.622} C_VEL
LIN {X 0,Y 191.134,Z 651.642,A -85,B 0,C 180,E1 -21788.991,E2 -21788.991} C_VEL
LIN {X 0,Y 191.989,Z 642.247,A -85,B 0,C 180,E1 -21792.688,E2 -21792.688} C_VEL
LIN {X 0,Y 193.142,Z 632.578,A -85,B 0,C 180,E1 -21795.838,E2 -21795.838} C_VEL
LIN {X 0,Y 194.68,Z 621.015,A -85,B 0,C 180,E1 -21798.96,E2 -21798.96} C_VEL
LIN {X 0,Y 196.412,Z 608.231,A -85,B 0,C 180,E1 -21801.791,E2 -21801.791} C_VEL
LIN {X 0,Y 198.375,Z 594.252,A -85,B 0,C 180,E1 -21804.321,E2 -21804.321} C_VEL
LIN {X 0,Y 200.214,Z 580.699,A -85,B 0,C 180,E1 -21806.306,E2 -21806.306} C_VEL
LIN {X 0,Y 201.906,Z 566.05,A -85,B 0,C 180,E1 -21808.029,E2 -21808.029} C_VEL
LIN {X 0,Y 203.421,Z 550.674,A -85,B 0,C 180,E1 -21809.423,E2 -21809.423} C_VEL
LIN {X 0,Y 205.11,Z 532.26,A -85,B 0,C 180,E1 -21810.786,E2 -21810.786} C_VEL
LIN {X 0,Y 205.782,Z 528.324,A -85,B 0,C 180,E1 -21811.317,E2 -21811.317} C_VEL
LIN {X 0,Y 207.29,Z 526.174,A -85,B 0,C 180,E1 -21811.986,E2 -21811.986} C_VEL
LIN {X 0,Y 209.116,Z 522.225,A -85,B 0,C 180,E1 -21812.53,E2 -21812.53} C_VEL
LIN {X 0,Y 212.76,Z 511.287,A -85,B 0,C 180,E1 -21813.381,E2 -21813.381} C_VEL
LIN {X 0,Y 217.694,Z 494.211,A -85,B 0,C 180,E1 -21814.33,E2 -21814.33} C_VEL
LIN {X 0,Y 218.485,Z 492.549,A -85,B 0,C 180,E1 -21814.538,E2 -21814.538} C_VEL
LIN {X 0,Y 221.011,Z 488.613,A -85,B 0,C 180,E1 -21815.258,E2 -21815.258} C_VEL
LIN {X 0,Y 223.894,Z 481.826,A -85,B 0,C 180,E1 -21815.923,E2 -21815.923} C_VEL
LIN {X 0,Y 227.743,Z 469.74,A -85,B 0,C 180,E1 -21816.613,E2 -21816.613} C_VEL
LIN {X 0,Y 230.975,Z 458.779,A -85,B 0,C 180,E1 -21817.125,E2 -21817.125} C_VEL
LIN {X 0,Y 234.019,Z 454.846,A -85,B 0,C 180,E1 -21817.904,E2 -21817.904} C_VEL
LIN {X 0,Y 236.725,Z 449.952,A -85,B 0,C 180,E1 -21818.501,E2 -21818.501} C_VEL
LIN {X 0,Y 242.351,Z 462.283,A -85,B 0,C 180,E1 -21820.69,E2 -21820.69} C_VEL
LIN {X 0,Y 244.373,Z 467.187,A -85,B 0,C 180,E1 -21821.45,E2 -21821.45} C_VEL
LIN {X 0,Y 238.886,Z 552.913,A -85,B 0,C 180,E1 -21823.728,E2 -21823.728} C_VEL
LIN {X 0,Y 237.445,Z 570.092,A -85,B 0,C 180,E1 -21824.282,E2 -21824.282} C_VEL
LIN {X 0,Y 235.207,Z 585.245,A -85,B 0,C 180,E1 -21825.02,E2 -21825.02} C_VEL
LIN {X 0,Y 232.27,Z 599.944,A -85,B 0,C 180,E1 -21826.049,E2 -21826.049} C_VEL
LIN {X 0,Y 228.596,Z 614.614,A -85,B 0,C 180,E1 -21827.439,E2 -21827.439} C_VEL
LIN {X 0,Y 224.459,Z 628.585,A -85,B 0,C 180,E1 -21829.185,E2 -21829.185} C_VEL
LIN {X 0,Y 219.932,Z 641.272,A -85,B 0,C 180,E1 -21831.161,E2 -21831.161} C_VEL
LIN {X 0,Y 215.342,Z 652.902,A -85,B 0,C 180,E1 -21833.443,E2 -21833.443} C_VEL
LIN {X 0,Y 210.734,Z 663.562,A -85,B 0,C 180,E1 -21836.04,E2 -21836.04} C_VEL
LIN {X 0,Y 206.582,Z 672.818,A -85,B 0,C 180,E1 -21838.84,E2 -21838.84} C_VEL
LIN {X 0,Y 202.314,Z 681.459,A -85,B 0,C 180,E1 -21842.033,E2 -21842.033} C_VEL
LIN {X 0,Y 198.216,Z 689.74,A -85,B 0,C 180,E1 -21845.936,E2 -21845.936} C_VEL
LIN {X 0,Y 195.012,Z 696.42,A -85,B 0,C 180,E1 -21850.011,E2 -21850.011} C_VEL
LIN {X 0,Y 192.703,Z 701.572,A -85,B 0,C 180,E1 -21854.125,E2 -21854.125} C_VEL
LIN {X 0,Y 191.439,Z 704.56,A -85,B 0,C 180,E1 -21857.275,E2 -21857.275} C_VEL
LIN {X 0,Y 190.461,Z 707.499,A -85,B 0,C 180,E1 -21861.512,E2 -21861.512} C_VEL
LIN {X 0,Y 190.086,Z 709.258,A -85,B 0,C 180,E1 -21865.759,E2 -21865.759} C_VEL
LIN {X 0,Y 190.115,Z 709.866,A -85,B 0,C 180,E1 -21870,E2 -21870} C_VEL
LIN {X 0,Y 190.086,Z 709.289,A -85,B 0,C 180,E1 -21874.24,E2 -21874.24} C_VEL
LIN {X 0,Y 190.46,Z 707.57,A -85,B 0,C 180,E1 -21878.488,E2 -21878.488} C_VEL
LIN {X 0,Y 191.428,Z 704.68,A -85,B 0,C 180,E1 -21882.725,E2 -21882.725} C_VEL
LIN {X 0,Y 193.19,Z 700.549,A -85,B 0,C 180,E1 -21886.919,E2 -21886.919} C_VEL
LIN {X 0,Y 195.633,Z 695.064,A -85,B 0,C 180,E1 -21891.054,E2 -21891.054} C_VEL
LIN {X 0,Y 199.101,Z 688.08,A -85,B 0,C 180,E1 -21895.061,E2 -21895.061} C_VEL
LIN {X 0,Y 202.81,Z 680.602,A -85,B 0,C 180,E1 -21898.456,E2 -21898.456} C_VEL
LIN {X 0,Y 207.032,Z 671.976,A -85,B 0,C 180,E1 -21901.593,E2 -21901.593} C_VEL
LIN {X 0,Y 211.35,Z 662.386,A -85,B 0,C 180,E1 -21904.423,E2 -21904.423} C_VEL
LIN {X 0,Y 216.486,Z 650.531,A -85,B 0,C 180,E1 -21907.203,E2 -21907.203} C_VEL
